LIN {X 0,Y 720.16,Z 195.522,A -85,B 0,C 180,E1 33617.616,E2 33617.616} C_VEL
LIN {X 0,Y 720.211,Z 195.516,A -85,B 0,C 180,E1 33614.811,E2 33614.811} C_VEL
LIN {X 0,Y 720.216,Z 195.521,A -85,B 0,C 180,E1 33611.789,E2 33611.789} C_VEL
LIN {X 0,Y 720.148,Z 195.522,A -85,B 0,C 180,E1 33609.077,E2 33609.077} C_VEL
LIN {X 0,Y 720.178,Z 195.522,A -85,B 0,C 180,E1 33605.959,E2 33605.959} C_VEL
LIN {X 0,Y 720.238,Z 195.651,A -85,B 0,C 180,E1 33604.404,E2 33604.404} C_VEL
LIN {X 0,Y 723.958,Z 206.616,A -85,B 0,C 180,E1 33603.441,E2 33603.441} C_VEL
LIN {X 0,Y 723.246,Z 247.825,A -85,B 0,C 180,E1 33600.537,E2 33600.537} C_VEL
LIN {X 0,Y 722.668,Z 288.727,A -85,B 0,C 180,E1 33597.748,E2 33597.748} C_VEL
LIN {X 0,Y 722.544,Z 304.623,A -85,B 0,C 180,E1 33596.701,E2 33596.701} C_VEL
LIN {X 0,Y 723.876,Z 312.314,A -85,B 0,C 180,E1 33596.564,E2 33596.564} C_VEL
LIN {X 0,Y 722.993,Z 604.896,A -85,B 0,C 180,E1 33593.438,E2 33593.438} C_VEL
LIN {X 0,Y 722.818,Z 626.619,A -85,B 0,C 180,E1 33593.09,E2 33593.09} C_VEL
LIN {X 0,Y 722.561,Z 650.13,A -85,B 0,C 180,E1 33592.539,E2 33592.539} C_VEL
LIN {X 0,Y 722.316,Z 669.51,A -85,B 0,C 180,E1 33591.948,E2 33591.948} C_VEL
LIN {X 0,Y 722.014,Z 689.697,A -85,B 0,C 180,E1 33591.189,E2 33591.189} C_VEL
LIN {X 0,Y 721.715,Z 710.059,A -85,B 0,C 180,E1 33590.265,E2 33590.265} C_VEL
LIN {X 0,Y 721.363,Z 729.936,A -85,B 0,C 180,E1 33589.178,E2 33589.178} C_VEL
LIN {X 0,Y 721.062,Z 746.81,A -85,B 0,C 180,E1 33588.097,E2 33588.097} C_VEL
LIN {X 0,Y 720.802,Z 763.918,A -85,B 0,C 180,E1 33586.83,E2 33586.83} C_VEL
LIN {X 0,Y 720.546,Z 779.819,A -85,B 0,C 180,E1 33585.452,E2 33585.452} C_VEL
LIN {X 0,Y 720.356,Z 792.902,A -85,B 0,C 180,E1 33584.14,E2 33584.14} C_VEL
LIN {X 0,Y 720.195,Z 806.207,A -85,B 0,C 180,E1 33582.59,E2 33582.59} C_VEL
LIN {X 0,Y 720.072,Z 817.974,A -85,B 0,C 180,E1 33580.965,E2 33580.965} C_VEL
LIN {X 0,Y 719.998,Z 827.271,A -85,B 0,C 180,E1 33579.432,E2 33579.432} C_VEL
LIN {X 0,Y 719.944,Z 835.631,A -85,B 0,C 180,E1 33577.742,E2 33577.742} C_VEL
LIN {X 0,Y 719.927,Z 842.505,A -85,B 0,C 180,E1 33575.979,E2 33575.979} C_VEL
LIN {X 0,Y 719.92,Z 847.512,A -85,B 0,C 180,E1 33574.221,E2 33574.221} C_VEL
LIN {X 0,Y 719.914,Z 850.607,A -85,B 0,C 180,E1 33572.547,E2 33572.547} C_VEL
LIN {X 0,Y 719.914,Z 852.289,A -85,B 0,C 180,E1 33570.796,E2 33570.796} C_VEL
LIN {X 0,Y 719.909,Z 852.219,A -85,B 0,C 180,E1 33568.965,E2 33568.965} C_VEL
LIN {X 0,Y 719.913,Z 850.51,A -85,B 0,C 180,E1 33567.293,E2 33567.293} C_VEL
LIN {X 0,Y 719.919,Z 847.147,A -85,B 0,C 180,E1 33565.539,E2 33565.539} C_VEL
LIN {X 0,Y 719.936,Z 841.735,A -85,B 0,C 180,E1 33563.701,E2 33563.701} C_VEL
LIN {X 0,Y 719.958,Z 834.828,A -85,B 0,C 180,E1 33561.985,E2 33561.985} C_VEL
LIN {X 0,Y 720.007,Z 826.408,A -85,B 0,C 180,E1 33560.326,E2 33560.326} C_VEL
LIN {X 0,Y 720.103,Z 815.862,A -85,B 0,C 180,E1 33558.628,E2 33558.628} C_VEL
LIN {X 0,Y 720.228,Z 804.11,A -85,B 0,C 180,E1 33557.056,E2 33557.056} C_VEL
LIN {X 0,Y 720.377,Z 791.433,A -85,B 0,C 180,E1 33555.614,E2 33555.614} C_VEL
LIN {X 0,Y 720.595,Z 776.326,A -85,B 0,C 180,E1 33554.136,E2 33554.136} C_VEL
LIN {X 0,Y 720.851,Z 759.998,A -85,B 0,C 180,E1 33552.774,E2 33552.774} C_VEL
LIN {X 0,Y 721.109,Z 744.471,A -85,B 0,C 180,E1 33551.654,E2 33551.654} C_VEL
LIN {X 0,Y 721.411,Z 726.463,A -85,B 0,C 180,E1 33550.529,E2 33550.529} C_VEL
LIN {X 0,Y 721.75,Z 706.47,A -85,B 0,C 180,E1 33549.474,E2 33549.474} C_VEL
LIN {X 0,Y 722.033,Z 688.563,A -85,B 0,C 180,E1 33548.675,E2 33548.675} C_VEL
LIN {X 0,Y 722.331,Z 668.395,A -85,B 0,C 180,E1 33547.925,E2 33547.925} C_VEL
LIN {X 0,Y 722.629,Z 645.716,A -85,B 0,C 180,E1 33547.254,E2 33547.254} C_VEL
LIN {X 0,Y 722.835,Z 624.224,A -85,B 0,C 180,E1 33546.776,E2 33546.776} C_VEL
LIN {X 0,Y 723.001,Z 603.601,A -85,B 0,C 180,E1 33546.455,E2 33546.455} C_VEL
LIN {X 0,Y 723.876,Z 312.433,A -85,B 0,C 180,E1 33543.347,E2 33543.347} C_VEL
LIN {X 0,Y 722.906,Z 306.324,A -85,B 0,C 180,E1 33543.242,E2 33543.242} C_VEL
LIN {X 0,Y 722.485,Z 303.913,A -85,B 0,C 180,E1 33543.181,E2 33543.181} C_VEL
LIN {X 0,Y 723.04,Z 261.674,A -85,B 0,C 180,E1 33540.325,E2 33540.325} C_VEL
LIN {X 0,Y 723.666,Z 220.838,A -85,B 0,C 180,E1 33537.488,E2 33537.488} C_VEL
LIN {X 0,Y 723.746,Z 206.018,A -85,B 0,C 180,E1 33536.416,E2 33536.416} C_VEL
LIN {X 0,Y 720.207,Z 195.519,A -85,B 0,C 180,E1 33535.473,E2 33535.473} C_VEL
LIN {X 0,Y 720.201,Z 195.524,A -85,B 0,C 180,E1 33532.548,E2 33532.548} C_VEL
LIN {X 0,Y 720.212,Z 195.511,A -85,B 0,C 180,E1 33529.478,E2 33529.478} C_VEL
LIN {X 0,Y 720.206,Z 195.521,A -85,B 0,C 180,E1 33526.479,E2 33526.479} C_VEL
LIN {X 0,Y 720.215,Z 195.509,A -85,B 0,C 180,E1 33523.411,E2 33523.411} C_VEL
LIN {X 0,Y 720.219,Z 195.519,A -85,B 0,C 180,E1 33520.343,E2 33520.343} C_VEL
LIN {X 0,Y 720.208,Z 195.509,A -85,B 0,C 180,E1 33517.252,E2 33517.252} C_VEL
LIN {X 0,Y 720.216,Z 195.521,A -85,B 0,C 180,E1 33514.305,E2 33514.305} C_VEL
LIN {X 0,Y 720.211,Z 195.51,A -85,B 0,C 180,E1 33511.217,E2 33511.217} C_VEL
LIN {X 0,Y 720.217,Z 195.517,A -85,B 0,C 180,E1 33508.166,E2 33508.166} C_VEL
LIN {X 0,Y 720.211,Z 195.51,A -85,B 0,C 180,E1 33505.14,E2 33505.14} C_VEL
LIN {X 0,Y 720.212,Z 195.52,A -85,B 0,C 180,E1 33502.101,E2 33502.101} C_VEL
LIN {X 0,Y 720.215,Z 195.507,A -85,B 0,C 180,E1 33499.126,E2 33499.126} C_VEL
LIN {X 0,Y 720.214,Z 195.52,A -85,B 0,C 180,E1 33496.112,E2 33496.112} C_VEL
LIN {X 0,Y 720.219,Z 195.506,A -85,B 0,C 180,E1 33493.079,E2 33493.079} C_VEL
LIN {X 0,Y 720.212,Z 195.52,A -85,B 0,C 180,E1 33490.075,E2 33490.075} C_VEL
LIN {X 0,Y 720.222,Z 195.506,A -85,B 0,C 180,E1 33487.098,E2 33487.098} C_VEL
LIN {X 0,Y 720.211,Z 195.521,A -85,B 0,C 180,E1 33484.06,E2 33484.06} C_VEL
LIN {X 0,Y 720.219,Z 195.508,A -85,B 0,C 180,E1 33481.034,E2 33481.034} C_VEL
LIN {X 0,Y 720.207,Z 195.52,A -85,B 0,C 180,E1 33478.011,E2 33478.011} C_VEL
LIN {X 0,Y 720.21,Z 195.51,A -85,B 0,C 180,E1 33475.062,E2 33475.062} C_VEL
LIN {X 0,Y 720.201,Z 195.518,A -85,B 0,C 180,E1 33471.939,E2 33471.939} C_VEL
LIN {X 0,Y 720.214,Z 195.51,A -85,B 0,C 180,E1 33468.954,E2 33468.954} C_VEL
LIN {X 0,Y 720.202,Z 195.52,A -85,B 0,C 180,E1 33465.939,E2 33465.939} C_VEL
LIN {X 0,Y 720.196,Z 195.512,A -85,B 0,C 180,E1 33463.049,E2 33463.049} C_VEL
LIN {X 0,Y 720.203,Z 195.521,A -85,B 0,C 180,E1 33459.945,E2 33459.945} C_VEL
LIN {X 0,Y 720.184,Z 195.514,A -85,B 0,C 180,E1 33457.123,E2 33457.123} C_VEL
LIN {X 0,Y 720.218,Z 195.522,A -85,B 0,C 180,E1 33454.109,E2 33454.109} C_VEL
LIN {X 0,Y 720.171,Z 195.516,A -85,B 0,C 180,E1 33451.289,E2 33451.289} C_VEL
LIN {X 0,Y 720.219,Z 195.515,A -85,B 0,C 180,E1 33448.44,E2 33448.44} C_VEL
LIN {X 0,Y 720.171,Z 195.519,A -85,B 0,C 180,E1 33445.559,E2 33445.559} C_VEL
LIN {X 0,Y 720.191,Z 195.514,A -85,B 0,C 180,E1 33442.837,E2 33442.837} C_VEL
LIN {X 0,Y 720.188,Z 195.522,A -85,B 0,C 180,E1 33439.783,E2 33439.783} C_VEL
LIN {X 0,Y 720.163,Z 195.518,A -85,B 0,C 180,E1 33437.131,E2 33437.131} C_VEL
LIN {X 0,Y 720.222,Z 195.518,A -85,B 0,C 180,E1 33434.244,E2 33434.244} C_VEL
LIN {X 0,Y 720.158,Z 195.522,A -85,B 0,C 180,E1 33431.368,E2 33431.368} C_VEL
LIN {X 0,Y 720.209,Z 195.663,A -85,B 0,C 180,E1 33429.793,E2 33429.793} C_VEL
LIN {X 0,Y 721.281,Z 198.701,A -85,B 0,C 180,E1 33429.577,E2 33429.577} C_VEL
LIN {X 0,Y 726.57,Z 209.646,A -85,B 0,C 180,E1 33428.712,E2 33428.712} C_VEL
LIN {X 0,Y 725.859,Z 260.94,A -85,B 0,C 180,E1 33426.323,E2 33426.323} C_VEL
LIN {X 0,Y 725.458,Z 299.229,A -85,B 0,C 180,E1 33424.598,E2 33424.598} C_VEL
LIN {X 0,Y 726.47,Z 307.17,A -85,B 0,C 180,E1 33424.45,E2 33424.45} C_VEL
LIN {X 0,Y 725.424,Z 570.263,A -85,B 0,C 180,E1 33421.465,E2 33421.465} C_VEL
LIN {X 0,Y 724.936,Z 690.96,A -85,B 0,C 180,E1 33420.101,E2 33420.101} C_VEL
LIN {X 0,Y 724.634,Z 716.508,A -85,B 0,C 180,E1 33419.668,E2 33419.668} C_VEL
LIN {X 0,Y 724.35,Z 738.123,A -85,B 0,C 180,E1 33419.168,E2 33419.168} C_VEL
LIN {X 0,Y 724.01,Z 761.286,A -85,B 0,C 180,E1 33418.499,E2 33418.499} C_VEL
LIN {X 0,Y 723.566,Z 783.363,A -85,B 0,C 180,E1 33417.711,E2 33417.711} C_VEL
LIN {X 0,Y 723.176,Z 805.236,A -85,B 0,C 180,E1 33416.791,E2 33416.791} C_VEL
LIN {X 0,Y 722.679,Z 827.148,A -85,B 0,C 180,E1 33415.706,E2 33415.706} C_VEL
LIN {X 0,Y 722.248,Z 847.62,A -85,B 0,C 180,E1 33414.54,E2 33414.54} C_VEL
LIN {X 0,Y 721.793,Z 867.842,A -85,B 0,C 180,E1 33413.211,E2 33413.211} C_VEL
LIN {X 0,Y 721.414,Z 886.71,A -85,B 0,C 180,E1 33411.805,E2 33411.805} C_VEL
LIN {X 0,Y 721.029,Z 904.462,A -85,B 0,C 180,E1 33410.285,E2 33410.285} C_VEL
LIN {X 0,Y 720.755,Z 920.964,A -85,B 0,C 180,E1 33408.691,E2 33408.691} C_VEL
LIN {X 0,Y 720.478,Z 935.22,A -85,B 0,C 180,E1 33407.111,E2 33407.111} C_VEL
LIN {X 0,Y 720.304,Z 948.442,A -85,B 0,C 180,E1 33405.458,E2 33405.458} C_VEL
LIN {X 0,Y 720.157,Z 960.276,A -85,B 0,C 180,E1 33403.734,E2 33403.734} C_VEL
LIN {X 0,Y 720.066,Z 970.03,A -85,B 0,C 180,E1 33402.104,E2 33402.104} C_VEL
LIN {X 0,Y 719.982,Z 980.182,A -85,B 0,C 180,E1 33400.078,E2 33400.078} C_VEL
LIN {X 0,Y 719.928,Z 986.815,A -85,B 0,C 180,E1 33398.466,E2 33398.466} C_VEL
LIN {X 0,Y 719.913,Z 993.245,A -85,B 0,C 180,E1 33396.54,E2 33396.54} C_VEL
LIN {X 0,Y 719.916,Z 997.813,A -85,B 0,C 180,E1 33394.62,E2 33394.62} C_VEL
LIN {X 0,Y 719.882,Z 1000.685,A -85,B 0,C 180,E1 33392.866,E2 33392.866} C_VEL
LIN {X 0,Y 719.891,Z 1002.262,A -85,B 0,C 180,E1 33390.875,E2 33390.875} C_VEL
LIN {X 0,Y 719.883,Z 1002.306,A -85,B 0,C 180,E1 33389.284,E2 33389.284} C_VEL
LIN {X 0,Y 719.888,Z 1001.017,A -85,B 0,C 180,E1 33387.373,E2 33387.373} C_VEL
LIN {X 0,Y 719.917,Z 997.971,A -85,B 0,C 180,E1 33385.459,E2 33385.459} C_VEL
LIN {X 0,Y 719.915,Z 993.864,A -85,B 0,C 180,E1 33383.701,E2 33383.701} C_VEL
LIN {X 0,Y 719.936,Z 987.422,A -85,B 0,C 180,E1 33381.695,E2 33381.695} C_VEL
LIN {X 0,Y 719.968,Z 980.892,A -85,B 0,C 180,E1 33380.084,E2 33380.084} C_VEL
LIN {X 0,Y 720.053,Z 971.867,A -85,B 0,C 180,E1 33378.221,E2 33378.221} C_VEL
LIN {X 0,Y 720.143,Z 961.081,A -85,B 0,C 180,E1 33376.392,E2 33376.392} C_VEL
LIN {X 0,Y 720.295,Z 949.06,A -85,B 0,C 180,E1 33374.625,E2 33374.625} C_VEL
LIN {X 0,Y 720.472,Z 935.927,A -85,B 0,C 180,E1 33372.972,E2 33372.972} C_VEL
LIN {X 0,Y 720.739,Z 921.74,A -85,B 0,C 180,E1 33371.393,E2 33371.393} C_VEL
LIN {X 0,Y 721.008,Z 905.39,A -85,B 0,C 180,E1 33369.799,E2 33369.799} C_VEL
LIN {X 0,Y 721.376,Z 888.27,A -85,B 0,C 180,E1 33368.322,E2 33368.322} C_VEL
LIN {X 0,Y 721.76,Z 869.107,A -85,B 0,C 180,E1 33366.879,E2 33366.879} C_VEL
LIN {X 0,Y 722.231,Z 849.066,A -85,B 0,C 180,E1 33365.547,E2 33365.547} C_VEL
LIN {X 0,Y 722.653,Z 827.944,A -85,B 0,C 180,E1 33364.337,E2 33364.337} C_VEL
LIN {X 0,Y 723.165,Z 806.229,A -85,B 0,C 180,E1 33363.253,E2 33363.253} C_VEL
LIN {X 0,Y 723.547,Z 784.481,A -85,B 0,C 180,E1 33362.333,E2 33362.333} C_VEL
LIN {X 0,Y 723.972,Z 762.568,A -85,B 0,C 180,E1 33361.544,E2 33361.544} C_VEL
LIN {X 0,Y 724.349,Z 738.334,A -85,B 0,C 180,E1 33360.838,E2 33360.838} C_VEL
LIN {X 0,Y 724.63,Z 716.764,A -85,B 0,C 180,E1 33360.337,E2 33360.337} C_VEL
LIN {X 0,Y 724.936,Z 691.166,A -85,B 0,C 180,E1 33359.902,E2 33359.902} C_VEL
LIN {X 0,Y 725.376,Z 582.637,A -85,B 0,C 180,E1 33358.674,E2 33358.674} C_VEL
LIN {X 0,Y 726.451,Z 311.994,A -85,B 0,C 180,E1 33355.606,E2 33355.606} C_VEL
LIN {X 0,Y 726.227,Z 304.001,A -85,B 0,C 180,E1 33355.5,E2 33355.5} C_VEL
LIN {X 0,Y 725.36,Z 298.429,A -85,B 0,C 180,E1 33355.382,E2 33355.382} C_VEL
LIN {X 0,Y 726.223,Z 237.623,A -85,B 0,C 180,E1 33352.602,E2 33352.602} C_VEL
LIN {X 0,Y 726.566,Z 209.659,A -85,B 0,C 180,E1 33351.288,E2 33351.288} C_VEL
LIN {X 0,Y 721.385,Z 198.876,A -85,B 0,C 180,E1 33350.413,E2 33350.413} C_VEL
LIN {X 0,Y 720.172,Z 195.526,A -85,B 0,C 180,E1 33350.156,E2 33350.156} C_VEL
LIN {X 0,Y 720.211,Z 195.521,A -85,B 0,C 180,E1 33347.142,E2 33347.142} C_VEL
LIN {X 0,Y 720.177,Z 195.524,A -85,B 0,C 180,E1 33344.296,E2 33344.296} C_VEL
LIN {X 0,Y 720.221,Z 195.519,A -85,B 0,C 180,E1 33341.316,E2 33341.316} C_VEL
LIN {X 0,Y 720.195,Z 195.524,A -85,B 0,C 180,E1 33338.332,E2 33338.332} C_VEL
LIN {X 0,Y 720.223,Z 195.521,A -85,B 0,C 180,E1 33335.375,E2 33335.375} C_VEL
LIN {X 0,Y 720.201,Z 195.528,A -85,B 0,C 180,E1 33333.906,E2 33333.906} C_VEL
LIN {X 0,Y 724.343,Z 207.121,A -85,B 0,C 180,E1 33332.948,E2 33332.948} C_VEL
LIN {X 0,Y 723.304,Z 257.17,A -85,B 0,C 180,E1 33330.074,E2 33330.074} C_VEL
LIN {X 0,Y 722.6,Z 315.269,A -85,B 0,C 180,E1 33326.859,E2 33326.859} C_VEL
LIN {X 0,Y 722.176,Z 369.58,A -85,B 0,C 180,E1 33323.933,E2 33323.933} C_VEL
LIN {X 0,Y 721.73,Z 424.416,A -85,B 0,C 180,E1 33321.028,E2 33321.028} C_VEL
LIN {X 0,Y 721.364,Z 470.562,A -85,B 0,C 180,E1 33318.625,E2 33318.625} C_VEL
LIN {X 0,Y 721.822,Z 478.064,A -85,B 0,C 180,E1 33318.535,E2 33318.535} C_VEL
LIN {X 0,Y 721.438,Z 679.938,A -85,B 0,C 180,E1 33316.459,E2 33316.459} C_VEL
LIN {X 0,Y 721.316,Z 699.052,A -85,B 0,C 180,E1 33316.11,E2 33316.11} C_VEL
LIN {X 0,Y 721.167,Z 717.241,A -85,B 0,C 180,E1 33315.629,E2 33315.629} C_VEL
LIN {X 0,Y 720.969,Z 734.998,A -85,B 0,C 180,E1 33315.008,E2 33315.008} C_VEL
LIN {X 0,Y 720.803,Z 751.994,A -85,B 0,C 180,E1 33314.254,E2 33314.254} C_VEL
LIN {X 0,Y 720.617,Z 767.716,A -85,B 0,C 180,E1 33313.398,E2 33313.398} C_VEL
LIN {X 0,Y 720.432,Z 783.102,A -85,B 0,C 180,E1 33312.382,E2 33312.382} C_VEL
LIN {X 0,Y 720.274,Z 796.852,A -85,B 0,C 180,E1 33311.288,E2 33311.288} C_VEL
LIN {X 0,Y 720.145,Z 809.523,A -85,B 0,C 180,E1 33310.076,E2 33310.076} C_VEL
LIN {X 0,Y 720.05,Z 820.643,A -85,B 0,C 180,E1 33308.786,E2 33308.786} C_VEL
LIN {X 0,Y 719.983,Z 830.232,A -85,B 0,C 180,E1 33307.421,E2 33307.421} C_VEL
LIN {X 0,Y 719.946,Z 837.854,A -85,B 0,C 180,E1 33306.059,E2 33306.059} C_VEL
LIN {X 0,Y 719.921,Z 844.045,A -85,B 0,C 180,E1 33304.621,E2 33304.621} C_VEL
LIN {X 0,Y 719.914,Z 848.466,A -85,B 0,C 180,E1 33303.185,E2 33303.185} C_VEL
LIN {X 0,Y 719.912,Z 851.34,A -85,B 0,C 180,E1 33301.671,E2 33301.671} C_VEL
LIN {X 0,Y 719.912,Z 852.449,A -85,B 0,C 180,E1 33300.159,E2 33300.159} C_VEL
LIN {X 0,Y 719.913,Z 851.819,A -85,B 0,C 180,E1 33298.647,E2 33298.647} C_VEL
LIN {X 0,Y 719.914,Z 849.435,A -85,B 0,C 180,E1 33297.134,E2 33297.134} C_VEL
LIN {X 0,Y 719.922,Z 845.232,A -85,B 0,C 180,E1 33295.619,E2 33295.619} C_VEL
LIN {X 0,Y 719.936,Z 839.461,A -85,B 0,C 180,E1 33294.181,E2 33294.181} C_VEL
LIN {X 0,Y 719.981,Z 831.802,A -85,B 0,C 180,E1 33292.74,E2 33292.74} C_VEL
LIN {X 0,Y 720.037,Z 822.605,A -85,B 0,C 180,E1 33291.374,E2 33291.374} C_VEL
LIN {X 0,Y 720.131,Z 811.918,A -85,B 0,C 180,E1 33290.086,E2 33290.086} C_VEL
LIN {X 0,Y 720.249,Z 799.731,A -85,B 0,C 180,E1 33288.874,E2 33288.874} C_VEL
LIN {X 0,Y 720.4,Z 785.987,A -85,B 0,C 180,E1 33287.739,E2 33287.739} C_VEL
LIN {X 0,Y 720.572,Z 771.146,A -85,B 0,C 180,E1 33286.721,E2 33286.721} C_VEL
LIN {X 0,Y 720.732,Z 758.498,A -85,B 0,C 180,E1 33285.987,E2 33285.987} C_VEL
LIN {X 0,Y 719.842,Z 752.168,A -85,B 0,C 180,E1 33285.636,E2 33285.636} C_VEL
LIN {X 0,Y 714.42,Z 736.944,A -85,B 0,C 180,E1 33284.836,E2 33284.836} C_VEL
LIN {X 0,Y 713.298,Z 730.158,A -85,B 0,C 180,E1 33284.548,E2 33284.548} C_VEL
LIN {X 0,Y 713.28,Z 729.152,A -85,B 0,C 180,E1 33284.511,E2 33284.511} C_VEL
LIN {X 0,Y 713.505,Z 710.535,A -85,B 0,C 180,E1 33283.911,E2 33283.911} C_VEL
LIN {X 0,Y 713.666,Z 691.674,A -85,B 0,C 180,E1 33283.468,E2 33283.468} C_VEL
LIN {X 0,Y 713.79,Z 672.625,A -85,B 0,C 180,E1 33283.177,E2 33283.177} C_VEL
LIN {X 0,Y 714.094,Z 473.867,A -85,B 0,C 180,E1 33281.121,E2 33281.121} C_VEL
LIN {X 0,Y 713.625,Z 469.588,A -85,B 0,C 180,E1 33281.045,E2 33281.045} C_VEL
LIN {X 0,Y 714.172,Z 418.046,A -85,B 0,C 180,E1 33278.308,E2 33278.308} C_VEL
LIN {X 0,Y 714.783,Z 362.685,A -85,B 0,C 180,E1 33275.319,E2 33275.319} C_VEL
LIN {X 0,Y 715.433,Z 312.1,A -85,B 0,C 180,E1 33272.535,E2 33272.535} C_VEL
LIN {X 0,Y 716.158,Z 259.687,A -85,B 0,C 180,E1 33269.599,E2 33269.599} C_VEL
LIN {X 0,Y 716.883,Z 210.15,A -85,B 0,C 180,E1 33266.76,E2 33266.76} C_VEL
LIN {X 0,Y 716.315,Z 207.723,A -85,B 0,C 180,E1 33266.589,E2 33266.589} C_VEL
LIN {X 0,Y 712.272,Z 196.512,A -85,B 0,C 180,E1 33265.693,E2 33265.693} C_VEL
LIN {X 0,Y 712.274,Z 196.504,A -85,B 0,C 180,E1 33262.667,E2 33262.667} C_VEL
LIN {X 0,Y 712.208,Z 196.513,A -85,B 0,C 180,E1 33259.773,E2 33259.773} C_VEL
LIN {X 0,Y 712.269,Z 196.511,A -85,B 0,C 180,E1 33257.09,E2 33257.09} C_VEL
LIN {X 0,Y 712.265,Z 196.505,A -85,B 0,C 180,E1 33254.131,E2 33254.131} C_VEL
LIN {X 0,Y 712.235,Z 196.508,A -85,B 0,C 180,E1 33251.286,E2 33251.286} C_VEL
LIN {X 0,Y 712.276,Z 196.512,A -85,B 0,C 180,E1 33248.434,E2 33248.434} C_VEL
LIN {X 0,Y 712.234,Z 196.514,A -85,B 0,C 180,E1 33245.536,E2 33245.536} C_VEL
LIN {X 0,Y 712.28,Z 196.515,A -85,B 0,C 180,E1 33244.793,E2 33244.793} C_VEL
LIN {X 0,Y 716.825,Z 210.095,A -85,B 0,C 180,E1 33243.583,E2 33243.583} C_VEL
LIN {X 0,Y 715.958,Z 248.509,A -85,B 0,C 180,E1 33240.834,E2 33240.834} C_VEL
LIN {X 0,Y 715.265,Z 289.395,A -85,B 0,C 180,E1 33238.015,E2 33238.015} C_VEL
LIN {X 0,Y 715.109,Z 304.617,A -85,B 0,C 180,E1 33237.001,E2 33237.001} C_VEL
LIN {X 0,Y 716.715,Z 313.568,A -85,B 0,C 180,E1 33236.837,E2 33236.837} C_VEL
LIN {X 0,Y 715.65,Z 604.587,A -85,B 0,C 180,E1 33233.698,E2 33233.698} C_VEL
LIN {X 0,Y 715.451,Z 625.147,A -85,B 0,C 180,E1 33233.369,E2 33233.369} C_VEL
LIN {X 0,Y 715.193,Z 647.921,A -85,B 0,C 180,E1 33232.85,E2 33232.85} C_VEL
LIN {X 0,Y 714.824,Z 669.791,A -85,B 0,C 180,E1 33232.18,E2 33232.18} C_VEL
LIN {X 0,Y 714.474,Z 689.691,A -85,B 0,C 180,E1 33231.424,E2 33231.424} C_VEL
LIN {X 0,Y 714.107,Z 710.089,A -85,B 0,C 180,E1 33230.489,E2 33230.489} C_VEL
LIN {X 0,Y 713.674,Z 729.931,A -85,B 0,C 180,E1 33229.393,E2 33229.393} C_VEL
LIN {X 0,Y 713.324,Z 746.817,A -85,B 0,C 180,E1 33228.3,E2 33228.3} C_VEL
LIN {X 0,Y 713.005,Z 763.646,A -85,B 0,C 180,E1 33227.043,E2 33227.043} C_VEL
LIN {X 0,Y 712.691,Z 779.818,A -85,B 0,C 180,E1 33225.627,E2 33225.627} C_VEL
LIN {X 0,Y 712.46,Z 792.9,A -85,B 0,C 180,E1 33224.3,E2 33224.3} C_VEL
LIN {X 0,Y 712.265,Z 806.215,A -85,B 0,C 180,E1 33222.733,E2 33222.733} C_VEL
LIN {X 0,Y 712.105,Z 818.482,A -85,B 0,C 180,E1 33221.009,E2 33221.009} C_VEL
LIN {X 0,Y 712.016,Z 827.705,A -85,B 0,C 180,E1 33219.457,E2 33219.457} C_VEL
LIN {X 0,Y 711.958,Z 835.635,A -85,B 0,C 180,E1 33217.83,E2 33217.83} C_VEL
LIN {X 0,Y 711.934,Z 842.509,A -85,B 0,C 180,E1 33216.047,E2 33216.047} C_VEL
LIN {X 0,Y 711.922,Z 847.507,A -85,B 0,C 180,E1 33214.269,E2 33214.269} C_VEL
LIN {X 0,Y 711.915,Z 850.608,A -85,B 0,C 180,E1 33212.576,E2 33212.576} C_VEL
LIN {X 0,Y 711.914,Z 852.292,A -85,B 0,C 180,E1 33210.805,E2 33210.805} C_VEL
LIN {X 0,Y 711.909,Z 852.214,A -85,B 0,C 180,E1 33208.954,E2 33208.954} C_VEL
LIN {X 0,Y 711.912,Z 850.509,A -85,B 0,C 180,E1 33207.263,E2 33207.263} C_VEL
LIN {X 0,Y 711.919,Z 847.149,A -85,B 0,C 180,E1 33205.489,E2 33205.489} C_VEL
LIN {X 0,Y 711.937,Z 841.731,A -85,B 0,C 180,E1 33203.63,E2 33203.63} C_VEL
LIN {X 0,Y 711.97,Z 834.967,A -85,B 0,C 180,E1 33201.927,E2 33201.927} C_VEL
LIN {X 0,Y 712.034,Z 826.408,A -85,B 0,C 180,E1 33200.217,E2 33200.217} C_VEL
LIN {X 0,Y 712.148,Z 815.858,A -85,B 0,C 180,E1 33198.5,E2 33198.5} C_VEL
LIN {X 0,Y 712.297,Z 804.33,A -85,B 0,C 180,E1 33196.938,E2 33196.938} C_VEL
LIN {X 0,Y 712.49,Z 791.429,A -85,B 0,C 180,E1 33195.451,E2 33195.451} C_VEL
LIN {X 0,Y 712.751,Z 776.122,A -85,B 0,C 180,E1 33193.938,E2 33193.938} C_VEL
LIN {X 0,Y 713.054,Z 760.059,A -85,B 0,C 180,E1 33192.585,E2 33192.585} C_VEL
LIN {X 0,Y 713.377,Z 744.454,A -85,B 0,C 180,E1 33191.448,E2 33191.448} C_VEL
LIN {X 0,Y 713.758,Z 726.057,A -85,B 0,C 180,E1 33190.288,E2 33190.288} C_VEL
LIN {X 0,Y 714.156,Z 705.733,A -85,B 0,C 180,E1 33189.211,E2 33189.211} C_VEL
LIN {X 0,Y 714.511,Z 687.71,A -85,B 0,C 180,E1 33188.405,E2 33188.405} C_VEL
LIN {X 0,Y 714.85,Z 668.384,A -85,B 0,C 180,E1 33187.681,E2 33187.681} C_VEL
LIN {X 0,Y 715.217,Z 645.269,A -85,B 0,C 180,E1 33186.994,E2 33186.994} C_VEL
LIN {X 0,Y 715.465,Z 624.006,A -85,B 0,C 180,E1 33186.52,E2 33186.52} C_VEL
LIN {X 0,Y 715.653,Z 604.059,A -85,B 0,C 180,E1 33186.206,E2 33186.206} C_VEL
LIN {X 0,Y 716.712,Z 314.22,A -85,B 0,C 180,E1 33183.08,E2 33183.08} C_VEL
LIN {X 0,Y 716.168,Z 309.757,A -85,B 0,C 180,E1 33183.008,E2 33183.008} C_VEL
LIN {X 0,Y 715.054,Z 303.905,A -85,B 0,C 180,E1 33182.88,E2 33182.88} C_VEL
LIN {X 0,Y 715.713,Z 262.054,A -85,B 0,C 180,E1 33180.018,E2 33180.018} C_VEL
LIN {X 0,Y 716.51,Z 225.81,A -85,B 0,C 180,E1 33177.446,E2 33177.446} C_VEL
LIN {X 0,Y 716.649,Z 209.27,A -85,B 0,C 180,E1 33176.26,E2 33176.26} C_VEL
LIN {X 0,Y 712.244,Z 196.513,A -85,B 0,C 180,E1 33175.087,E2 33175.087} C_VEL
LIN {X 0,Y 712.279,Z 196.512,A -85,B 0,C 180,E1 33172.217,E2 33172.217} C_VEL
LIN {X 0,Y 712.256,Z 196.503,A -85,B 0,C 180,E1 33169.248,E2 33169.248} C_VEL
LIN {X 0,Y 712.28,Z 196.508,A -85,B 0,C 180,E1 33166.299,E2 33166.299} C_VEL
LIN {X 0,Y 712.26,Z 196.5,A -85,B 0,C 180,E1 33163.232,E2 33163.232} C_VEL
LIN {X 0,Y 712.281,Z 196.507,A -85,B 0,C 180,E1 33160.222,E2 33160.222} C_VEL
LIN {X 0,Y 712.268,Z 196.498,A -85,B 0,C 180,E1 33157.232,E2 33157.232} C_VEL
LIN {X 0,Y 712.277,Z 196.508,A -85,B 0,C 180,E1 33154.225,E2 33154.225} C_VEL
LIN {X 0,Y 712.271,Z 196.5,A -85,B 0,C 180,E1 33151.199,E2 33151.199} C_VEL
LIN {X 0,Y 712.276,Z 196.506,A -85,B 0,C 180,E1 33148.143,E2 33148.143} C_VEL
LIN {X 0,Y 712.269,Z 196.499,A -85,B 0,C 180,E1 33145.084,E2 33145.084} C_VEL
LIN {X 0,Y 712.273,Z 196.509,A -85,B 0,C 180,E1 33142.1,E2 33142.1} C_VEL
LIN {X 0,Y 712.274,Z 196.496,A -85,B 0,C 180,E1 33139.092,E2 33139.092} C_VEL
LIN {X 0,Y 712.27,Z 196.508,A -85,B 0,C 180,E1 33136.055,E2 33136.055} C_VEL
LIN {X 0,Y 712.277,Z 196.495,A -85,B 0,C 180,E1 33133.035,E2 33133.035} C_VEL
LIN {X 0,Y 712.268,Z 196.509,A -85,B 0,C 180,E1 33130.025,E2 33130.025} C_VEL
LIN {X 0,Y 712.279,Z 196.496,A -85,B 0,C 180,E1 33127.015,E2 33127.015} C_VEL
LIN {X 0,Y 712.263,Z 196.508,A -85,B 0,C 180,E1 33123.944,E2 33123.944} C_VEL
LIN {X 0,Y 712.282,Z 196.497,A -85,B 0,C 180,E1 33120.965,E2 33120.965} C_VEL
LIN {X 0,Y 712.26,Z 196.507,A -85,B 0,C 180,E1 33117.908,E2 33117.908} C_VEL
LIN {X 0,Y 712.278,Z 196.499,A -85,B 0,C 180,E1 33114.926,E2 33114.926} C_VEL
LIN {X 0,Y 712.262,Z 196.507,A -85,B 0,C 180,E1 33111.93,E2 33111.93} C_VEL
LIN {X 0,Y 712.271,Z 196.5,A -85,B 0,C 180,E1 33108.994,E2 33108.994} C_VEL
LIN {X 0,Y 712.263,Z 196.509,A -85,B 0,C 180,E1 33105.94,E2 33105.94} C_VEL
LIN {X 0,Y 712.261,Z 196.501,A -85,B 0,C 180,E1 33103.022,E2 33103.022} C_VEL
LIN {X 0,Y 712.258,Z 196.509,A -85,B 0,C 180,E1 33099.883,E2 33099.883} C_VEL
LIN {X 0,Y 712.252,Z 196.503,A -85,B 0,C 180,E1 33097.029,E2 33097.029} C_VEL
LIN {X 0,Y 712.265,Z 196.508,A -85,B 0,C 180,E1 33093.935,E2 33093.935} C_VEL
LIN {X 0,Y 712.238,Z 196.503,A -85,B 0,C 180,E1 33091.123,E2 33091.123} C_VEL
LIN {X 0,Y 712.281,Z 196.508,A -85,B 0,C 180,E1 33088.135,E2 33088.135} C_VEL
LIN {X 0,Y 712.228,Z 196.507,A -85,B 0,C 180,E1 33085.349,E2 33085.349} C_VEL
LIN {X 0,Y 712.281,Z 196.504,A -85,B 0,C 180,E1 33082.48,E2 33082.48} C_VEL
LIN {X 0,Y 712.23,Z 196.51,A -85,B 0,C 180,E1 33079.544,E2 33079.544} C_VEL
LIN {X 0,Y 712.251,Z 196.505,A -85,B 0,C 180,E1 33076.769,E2 33076.769} C_VEL
LIN {X 0,Y 712.24,Z 196.514,A -85,B 0,C 180,E1 33073.686,E2 33073.686} C_VEL
LIN {X 0,Y 712.22,Z 196.51,A -85,B 0,C 180,E1 33071.071,E2 33071.071} C_VEL
LIN {X 0,Y 712.307,Z 196.683,A -85,B 0,C 180,E1 33070.259,E2 33070.259} C_VEL
LIN {X 0,Y 713.368,Z 199.645,A -85,B 0,C 180,E1 33070.043,E2 33070.043} C_VEL
LIN {X 0,Y 719.946,Z 213.509,A -85,B 0,C 180,E1 33068.945,E2 33068.945} C_VEL
LIN {X 0,Y 719.057,Z 267.233,A -85,B 0,C 180,E1 33066.425,E2 33066.425} C_VEL
LIN {X 0,Y 718.641,Z 299.284,A -85,B 0,C 180,E1 33064.973,E2 33064.973} C_VEL
LIN {X 0,Y 719.861,Z 308.443,A -85,B 0,C 180,E1 33064.797,E2 33064.797} C_VEL
LIN {X 0,Y 718.584,Z 572.549,A -85,B 0,C 180,E1 33061.773,E2 33061.773} C_VEL
LIN {X 0,Y 718.004,Z 691.175,A -85,B 0,C 180,E1 33060.419,E2 33060.419} C_VEL
LIN {X 0,Y 717.648,Z 716.767,A -85,B 0,C 180,E1 33059.981,E2 33059.981} C_VEL
LIN {X 0,Y 717.298,Z 738.46,A -85,B 0,C 180,E1 33059.474,E2 33059.474} C_VEL
LIN {X 0,Y 716.853,Z 762.568,A -85,B 0,C 180,E1 33058.765,E2 33058.765} C_VEL
LIN {X 0,Y 716.339,Z 784.486,A -85,B 0,C 180,E1 33057.969,E2 33057.969} C_VEL
LIN {X 0,Y 715.831,Z 807.582,A -85,B 0,C 180,E1 33056.978,E2 33056.978} C_VEL
LIN {X 0,Y 715.246,Z 828.756,A -85,B 0,C 180,E1 33055.904,E2 33055.904} C_VEL
LIN {X 0,Y 714.719,Z 849.755,A -85,B 0,C 180,E1 33054.683,E2 33054.683} C_VEL
LIN {X 0,Y 714.182,Z 869.143,A -85,B 0,C 180,E1 33053.379,E2 33053.379} C_VEL
LIN {X 0,Y 713.72,Z 887.819,A -85,B 0,C 180,E1 33051.961,E2 33051.961} C_VEL
LIN {X 0,Y 713.298,Z 904.462,A -85,B 0,C 180,E1 33050.515,E2 33050.515} C_VEL
LIN {X 0,Y 712.937,Z 920.965,A -85,B 0,C 180,E1 33048.904,E2 33048.904} C_VEL
LIN {X 0,Y 712.616,Z 935.222,A -85,B 0,C 180,E1 33047.305,E2 33047.305} C_VEL
LIN {X 0,Y 712.389,Z 949.06,A -85,B 0,C 180,E1 33045.55,E2 33045.55} C_VEL
LIN {X 0,Y 712.21,Z 960.797,A -85,B 0,C 180,E1 33043.808,E2 33043.808} C_VEL
LIN {X 0,Y 712.093,Z 970.948,A -85,B 0,C 180,E1 33042.077,E2 33042.077} C_VEL
LIN {X 0,Y 711.997,Z 980.538,A -85,B 0,C 180,E1 33040.11,E2 33040.11} C_VEL
LIN {X 0,Y 711.935,Z 987.12,A -85,B 0,C 180,E1 33038.48,E2 33038.48} C_VEL
LIN {X 0,Y 711.916,Z 993.451,A -85,B 0,C 180,E1 33036.532,E2 33036.532} C_VEL
LIN {X 0,Y 711.913,Z 997.814,A -85,B 0,C 180,E1 33034.673,E2 33034.673} C_VEL
LIN {X 0,Y 711.882,Z 1000.685,A -85,B 0,C 180,E1 33032.898,E2 33032.898} C_VEL
LIN {X 0,Y 711.891,Z 1002.262,A -85,B 0,C 180,E1 33030.885,E2 33030.885} C_VEL
LIN {X 0,Y 711.883,Z 1002.306,A -85,B 0,C 180,E1 33029.276,E2 33029.276} C_VEL
LIN {X 0,Y 711.887,Z 1001.017,A -85,B 0,C 180,E1 33027.343,E2 33027.343} C_VEL
LIN {X 0,Y 711.917,Z 997.972,A -85,B 0,C 180,E1 33025.408,E2 33025.408} C_VEL
LIN {X 0,Y 711.915,Z 993.864,A -85,B 0,C 180,E1 33023.63,E2 33023.63} C_VEL
LIN {X 0,Y 711.937,Z 987.423,A -85,B 0,C 180,E1 33021.601,E2 33021.601} C_VEL
LIN {X 0,Y 711.989,Z 980.892,A -85,B 0,C 180,E1 33019.971,E2 33019.971} C_VEL
LIN {X 0,Y 712.085,Z 971.866,A -85,B 0,C 180,E1 33018.088,E2 33018.088} C_VEL
LIN {X 0,Y 712.2,Z 961.318,A -85,B 0,C 180,E1 33016.275,E2 33016.275} C_VEL
LIN {X 0,Y 712.375,Z 949.642,A -85,B 0,C 180,E1 33014.533,E2 33014.533} C_VEL
LIN {X 0,Y 712.602,Z 935.929,A -85,B 0,C 180,E1 33012.778,E2 33012.778} C_VEL
LIN {X 0,Y 712.922,Z 921.741,A -85,B 0,C 180,E1 33011.181,E2 33011.181} C_VEL
LIN {X 0,Y 713.27,Z 905.39,A -85,B 0,C 180,E1 33009.57,E2 33009.57} C_VEL
LIN {X 0,Y 713.688,Z 888.776,A -85,B 0,C 180,E1 33008.119,E2 33008.119} C_VEL
LIN {X 0,Y 714.166,Z 869.652,A -85,B 0,C 180,E1 33006.658,E2 33006.658} C_VEL
LIN {X 0,Y 714.698,Z 850.418,A -85,B 0,C 180,E1 33005.36,E2 33005.36} C_VEL
LIN {X 0,Y 715.218,Z 829.552,A -85,B 0,C 180,E1 33004.139,E2 33004.139} C_VEL
LIN {X 0,Y 715.786,Z 808.975,A -85,B 0,C 180,E1 33003.089,E2 33003.089} C_VEL
LIN {X 0,Y 716.313,Z 785.727,A -85,B 0,C 180,E1 33002.08,E2 33002.08} C_VEL
LIN {X 0,Y 716.771,Z 765.133,A -85,B 0,C 180,E1 33001.322,E2 33001.322} C_VEL
LIN {X 0,Y 717.283,Z 740.116,A -85,B 0,C 180,E1 33000.57,E2 33000.57} C_VEL
LIN {X 0,Y 717.613,Z 718.69,A -85,B 0,C 180,E1 33000.06,E2 33000.06} C_VEL
LIN {X 0,Y 717.992,Z 693.629,A -85,B 0,C 180,E1 32999.614,E2 32999.614} C_VEL
LIN {X 0,Y 718.269,Z 642.02,A -85,B 0,C 180,E1 32999.009,E2 32999.009} C_VEL
LIN {X 0,Y 719.445,Z 392.284,A -85,B 0,C 180,E1 32996.173,E2 32996.173} C_VEL
LIN {X 0,Y 719.68,Z 305.755,A -85,B 0,C 180,E1 32995.161,E2 32995.161} C_VEL
LIN {X 0,Y 718.539,Z 298.171,A -85,B 0,C 180,E1 32994.993,E2 32994.993} C_VEL
LIN {X 0,Y 719.603,Z 236.709,A -85,B 0,C 180,E1 32992.154,E2 32992.154} C_VEL
LIN {X 0,Y 719.965,Z 213.374,A -85,B 0,C 180,E1 32991.054,E2 32991.054} C_VEL
LIN {X 0,Y 713.431,Z 199.808,A -85,B 0,C 180,E1 32989.928,E2 32989.928} C_VEL
LIN {X 0,Y 712.281,Z 196.511,A -85,B 0,C 180,E1 32989.664,E2 32989.664} C_VEL
LIN {X 0,Y 712.279,Z 196.511,A -85,B 0,C 180,E1 32986.76,E2 32986.76} C_VEL
LIN {X 0,Y 712.282,Z 196.51,A -85,B 0,C 180,E1 32983.794,E2 32983.794} C_VEL
LIN {X 0,Y 712.264,Z 196.512,A -85,B 0,C 180,E1 32980.829,E2 32980.829} C_VEL
LIN {X 0,Y 712.28,Z 196.51,A -85,B 0,C 180,E1 32977.914,E2 32977.914} C_VEL
LIN {X 0,Y 712.252,Z 196.514,A -85,B 0,C 180,E1 32974.931,E2 32974.931} C_VEL
LIN {X 0,Y 712.253,Z 196.683,A -85,B 0,C 180,E1 32974.345,E2 32974.345} C_VEL
LIN {X 0,Y 717.389,Z 210.124,A -85,B 0,C 180,E1 32973.166,E2 32973.166} C_VEL
LIN {X 0,Y 716.102,Z 258.891,A -85,B 0,C 180,E1 32970.316,E2 32970.316} C_VEL
LIN {X 0,Y 715.192,Z 315.897,A -85,B 0,C 180,E1 32967.115,E2 32967.115} C_VEL
LIN {X 0,Y 714.624,Z 369.984,A -85,B 0,C 180,E1 32964.163,E2 32964.163} C_VEL
LIN {X 0,Y 714.076,Z 424.961,A -85,B 0,C 180,E1 32961.221,E2 32961.221} C_VEL
LIN {X 0,Y 713.69,Z 470.224,A -85,B 0,C 180,E1 32958.853,E2 32958.853} C_VEL
LIN {X 0,Y 714.267,Z 478.095,A -85,B 0,C 180,E1 32958.747,E2 32958.747} C_VEL
LIN {X 0,Y 713.764,Z 680.017,A -85,B 0,C 180,E1 32956.64,E2 32956.64} C_VEL
LIN {X 0,Y 713.62,Z 699.074,A -85,B 0,C 180,E1 32956.288,E2 32956.288} C_VEL
LIN {X 0,Y 713.437,Z 717.391,A -85,B 0,C 180,E1 32955.799,E2 32955.799} C_VEL
LIN {X 0,Y 713.216,Z 734.446,A -85,B 0,C 180,E1 32955.199,E2 32955.199} C_VEL
LIN {X 0,Y 713.007,Z 751.19,A -85,B 0,C 180,E1 32954.455,E2 32954.455} C_VEL
LIN {X 0,Y 712.784,Z 767.054,A -85,B 0,C 180,E1 32953.59,E2 32953.59} C_VEL
LIN {X 0,Y 712.567,Z 781.997,A -85,B 0,C 180,E1 32952.603,E2 32952.603} C_VEL
LIN {X 0,Y 712.373,Z 795.932,A -85,B 0,C 180,E1 32951.497,E2 32951.497} C_VEL
LIN {X 0,Y 712.209,Z 808.757,A -85,B 0,C 180,E1 32950.271,E2 32950.271} C_VEL
LIN {X 0,Y 712.087,Z 820.011,A -85,B 0,C 180,E1 32948.967,E2 32948.967} C_VEL
LIN {X 0,Y 712.002,Z 829.721,A -85,B 0,C 180,E1 32947.586,E2 32947.586} C_VEL
LIN {X 0,Y 711.952,Z 837.452,A -85,B 0,C 180,E1 32946.208,E2 32946.208} C_VEL
LIN {X 0,Y 711.927,Z 843.746,A -85,B 0,C 180,E1 32944.753,E2 32944.753} C_VEL
LIN {X 0,Y 711.914,Z 848.468,A -85,B 0,C 180,E1 32943.221,E2 32943.221} C_VEL
LIN {X 0,Y 711.913,Z 851.342,A -85,B 0,C 180,E1 32941.69,E2 32941.69} C_VEL
LIN {X 0,Y 711.913,Z 852.449,A -85,B 0,C 180,E1 32940.161,E2 32940.161} C_VEL
LIN {X 0,Y 711.912,Z 851.818,A -85,B 0,C 180,E1 32938.632,E2 32938.632} C_VEL
LIN {X 0,Y 711.915,Z 849.433,A -85,B 0,C 180,E1 32937.102,E2 32937.102} C_VEL
LIN {X 0,Y 711.923,Z 845.485,A -85,B 0,C 180,E1 32935.65,E2 32935.65} C_VEL
LIN {X 0,Y 711.94,Z 839.812,A -85,B 0,C 180,E1 32934.196,E2 32934.196} C_VEL
LIN {X 0,Y 711.987,Z 832.719,A -85,B 0,C 180,E1 32932.82,E2 32932.82} C_VEL
LIN {X 0,Y 712.053,Z 823.755,A -85,B 0,C 180,E1 32931.44,E2 32931.44} C_VEL
LIN {X 0,Y 712.161,Z 813.333,A -85,B 0,C 180,E1 32930.137,E2 32930.137} C_VEL
LIN {X 0,Y 712.307,Z 801.092,A -85,B 0,C 180,E1 32928.876,E2 32928.876} C_VEL
LIN {X 0,Y 712.491,Z 787.609,A -85,B 0,C 180,E1 32927.725,E2 32927.725} C_VEL
LIN {X 0,Y 712.703,Z 772.501,A -85,B 0,C 180,E1 32926.657,E2 32926.657} C_VEL
LIN {X 0,Y 712.932,Z 756.541,A -85,B 0,C 180,E1 32925.727,E2 32925.727} C_VEL
LIN {X 0,Y 713.137,Z 739.631,A -85,B 0,C 180,E1 32924.925,E2 32924.925} C_VEL
LIN {X 0,Y 713.28,Z 729.152,A -85,B 0,C 180,E1 32924.511,E2 32924.511} C_VEL
LIN {X 0,Y 712.665,Z 723.159,A -85,B 0,C 180,E1 32924.281,E2 32924.281} C_VEL
LIN {X 0,Y 707.093,Z 705.636,A -85,B 0,C 180,E1 32923.621,E2 32923.621} C_VEL
LIN {X 0,Y 705.967,Z 698.377,A -85,B 0,C 180,E1 32923.421,E2 32923.421} C_VEL
LIN {X 0,Y 705.952,Z 697.308,A -85,B 0,C 180,E1 32923.397,E2 32923.397} C_VEL
LIN {X 0,Y 706.113,Z 677.939,A -85,B 0,C 180,E1 32923.054,E2 32923.054} C_VEL
LIN {X 0,Y 706.629,Z 474.731,A -85,B 0,C 180,E1 32920.895,E2 32920.895} C_VEL
LIN {X 0,Y 705.964,Z 468.931,A -85,B 0,C 180,E1 32920.795,E2 32920.795} C_VEL
LIN {X 0,Y 706.627,Z 415.892,A -85,B 0,C 180,E1 32917.947,E2 32917.947} C_VEL
LIN {X 0,Y 707.369,Z 358.655,A -85,B 0,C 180,E1 32914.819,E2 32914.819} C_VEL
LIN {X 0,Y 708.094,Z 310.205,A -85,B 0,C 180,E1 32912.125,E2 32912.125} C_VEL
LIN {X 0,Y 708.987,Z 256.994,A -85,B 0,C 180,E1 32909.112,E2 32909.112} C_VEL
LIN {X 0,Y 709.718,Z 212.196,A -85,B 0,C 180,E1 32906.516,E2 32906.516} C_VEL
LIN {X 0,Y 704.332,Z 197.5,A -85,B 0,C 180,E1 32905.35,E2 32905.35} C_VEL
LIN {X 0,Y 704.344,Z 197.496,A -85,B 0,C 180,E1 32902.379,E2 32902.379} C_VEL
LIN {X 0,Y 704.266,Z 197.502,A -85,B 0,C 180,E1 32899.546,E2 32899.546} C_VEL
LIN {X 0,Y 704.345,Z 197.496,A -85,B 0,C 180,E1 32896.711,E2 32896.711} C_VEL
LIN {X 0,Y 704.333,Z 197.499,A -85,B 0,C 180,E1 32893.731,E2 32893.731} C_VEL
LIN {X 0,Y 704.305,Z 197.495,A -85,B 0,C 180,E1 32890.826,E2 32890.826} C_VEL
LIN {X 0,Y 704.268,Z 197.504,A -85,B 0,C 180,E1 32887.728,E2 32887.728} C_VEL
LIN {X 0,Y 704.339,Z 197.652,A -85,B 0,C 180,E1 32885.182,E2 32885.182} C_VEL
LIN {X 0,Y 709.779,Z 213.038,A -85,B 0,C 180,E1 32883.782,E2 32883.782} C_VEL
LIN {X 0,Y 708.933,Z 248.718,A -85,B 0,C 180,E1 32881.22,E2 32881.22} C_VEL
LIN {X 0,Y 708.094,Z 278.852,A -85,B 0,C 180,E1 32879.062,E2 32879.062} C_VEL
LIN {X 0,Y 707.707,Z 304.681,A -85,B 0,C 180,E1 32877.307,E2 32877.307} C_VEL
LIN {X 0,Y 709.572,Z 314.84,A -85,B 0,C 180,E1 32877.116,E2 32877.116} C_VEL
LIN {X 0,Y 708.323,Z 604.176,A -85,B 0,C 180,E1 32873.963,E2 32873.963} C_VEL
LIN {X 0,Y 708.111,Z 623.549,A -85,B 0,C 180,E1 32873.656,E2 32873.656} C_VEL
LIN {X 0,Y 707.825,Z 644.177,A -85,B 0,C 180,E1 32873.198,E2 32873.198} C_VEL
LIN {X 0,Y 707.416,Z 667.036,A -85,B 0,C 180,E1 32872.522,E2 32872.522} C_VEL
LIN {X 0,Y 707.008,Z 686.572,A -85,B 0,C 180,E1 32871.792,E2 32871.792} C_VEL
LIN {X 0,Y 706.609,Z 704.141,A -85,B 0,C 180,E1 32871.008,E2 32871.008} C_VEL
LIN {X 0,Y 706.199,Z 722.741,A -85,B 0,C 180,E1 32870.038,E2 32870.038} C_VEL
LIN {X 0,Y 705.716,Z 742.117,A -85,B 0,C 180,E1 32868.834,E2 32868.834} C_VEL
LIN {X 0,Y 705.32,Z 758.277,A -85,B 0,C 180,E1 32867.661,E2 32867.661} C_VEL
LIN {X 0,Y 704.961,Z 774.409,A -85,B 0,C 180,E1 32866.31,E2 32866.31} C_VEL
LIN {X 0,Y 704.623,Z 790.595,A -85,B 0,C 180,E1 32864.715,E2 32864.715} C_VEL
LIN {X 0,Y 704.384,Z 802.926,A -85,B 0,C 180,E1 32863.295,E2 32863.295} C_VEL
LIN {X 0,Y 704.202,Z 814.074,A -85,B 0,C 180,E1 32861.798,E2 32861.798} C_VEL
LIN {X 0,Y 704.077,Z 824.984,A -85,B 0,C 180,E1 32860.06,E2 32860.06} C_VEL
LIN {X 0,Y 703.991,Z 833.448,A -85,B 0,C 180,E1 32858.412,E2 32858.412} C_VEL
LIN {X 0,Y 703.935,Z 839.935,A -85,B 0,C 180,E1 32856.838,E2 32856.838} C_VEL
LIN {X 0,Y 703.916,Z 845.471,A -85,B 0,C 180,E1 32855.134,E2 32855.134} C_VEL
LIN {X 0,Y 703.903,Z 849.66,A -85,B 0,C 180,E1 32853.257,E2 32853.257} C_VEL
LIN {X 0,Y 703.9,Z 851.844,A -85,B 0,C 180,E1 32851.465,E2 32851.465} C_VEL
LIN {X 0,Y 703.902,Z 852.452,A -85,B 0,C 180,E1 32849.674,E2 32849.674} C_VEL
LIN {X 0,Y 703.911,Z 851.29,A -85,B 0,C 180,E1 32847.802,E2 32847.802} C_VEL
LIN {X 0,Y 703.919,Z 848.414,A -85,B 0,C 180,E1 32846.009,E2 32846.009} C_VEL
LIN {X 0,Y 703.925,Z 843.802,A -85,B 0,C 180,E1 32844.212,E2 32844.212} C_VEL
LIN {X 0,Y 703.954,Z 837.441,A -85,B 0,C 180,E1 32842.409,E2 32842.409} C_VEL
LIN {X 0,Y 704.021,Z 829.494,A -85,B 0,C 180,E1 32840.682,E2 32840.682} C_VEL
LIN {X 0,Y 704.122,Z 820.083,A -85,B 0,C 180,E1 32839.031,E2 32839.031} C_VEL
LIN {X 0,Y 704.287,Z 809.445,A -85,B 0,C 180,E1 32837.454,E2 32837.454} C_VEL
LIN {X 0,Y 704.516,Z 795.925,A -85,B 0,C 180,E1 32835.78,E2 32835.78} C_VEL
LIN {X 0,Y 704.779,Z 782.443,A -85,B 0,C 180,E1 32834.362,E2 32834.362} C_VEL
LIN {X 0,Y 705.124,Z 767.259,A -85,B 0,C 180,E1 32832.973,E2 32832.973} C_VEL
LIN {X 0,Y 705.535,Z 749.3,A -85,B 0,C 180,E1 32831.577,E2 32831.577} C_VEL
LIN {X 0,Y 705.94,Z 732.752,A -85,B 0,C 180,E1 32830.472,E2 32830.472} C_VEL
LIN {X 0,Y 706.371,Z 714.967,A -85,B 0,C 180,E1 32829.448,E2 32829.448} C_VEL
LIN {X 0,Y 706.858,Z 693.799,A -85,B 0,C 180,E1 32828.421,E2 32828.421} C_VEL
LIN {X 0,Y 707.285,Z 673.767,A -85,B 0,C 180,E1 32827.624,E2 32827.624} C_VEL
LIN {X 0,Y 707.599,Z 655.35,A -85,B 0,C 180,E1 32827.023,E2 32827.023} C_VEL
LIN {X 0,Y 707.945,Z 636.235,A -85,B 0,C 180,E1 32826.52,E2 32826.52} C_VEL
LIN {X 0,Y 708.226,Z 614.339,A -85,B 0,C 180,E1 32826.088,E2 32826.088} C_VEL
LIN {X 0,Y 708.439,Z 584.242,A -85,B 0,C 180,E1 32825.717,E2 32825.717} C_VEL
LIN {X 0,Y 709.568,Z 313.73,A -85,B 0,C 180,E1 32822.782,E2 32822.782} C_VEL
LIN {X 0,Y 707.643,Z 303.896,A -85,B 0,C 180,E1 32822.572,E2 32822.572} C_VEL
LIN {X 0,Y 708.447,Z 263.895,A -85,B 0,C 180,E1 32819.791,E2 32819.791} C_VEL
LIN {X 0,Y 709.423,Z 230.579,A -85,B 0,C 180,E1 32817.377,E2 32817.377} C_VEL
LIN {X 0,Y 709.669,Z 212.635,A -85,B 0,C 180,E1 32816.086,E2 32816.086} C_VEL
LIN {X 0,Y 704.312,Z 197.503,A -85,B 0,C 180,E1 32814.704,E2 32814.704} C_VEL
LIN {X 0,Y 704.342,Z 197.493,A -85,B 0,C 180,E1 32811.657,E2 32811.657} C_VEL
LIN {X 0,Y 704.315,Z 197.496,A -85,B 0,C 180,E1 32808.678,E2 32808.678} C_VEL
LIN {X 0,Y 704.337,Z 197.493,A -85,B 0,C 180,E1 32805.684,E2 32805.684} C_VEL
LIN {X 0,Y 704.312,Z 197.494,A -85,B 0,C 180,E1 32802.735,E2 32802.735} C_VEL
LIN {X 0,Y 704.329,Z 197.494,A -85,B 0,C 180,E1 32799.823,E2 32799.823} C_VEL
LIN {X 0,Y 704.314,Z 197.491,A -85,B 0,C 180,E1 32796.907,E2 32796.907} C_VEL
LIN {X 0,Y 704.33,Z 197.492,A -85,B 0,C 180,E1 32793.997,E2 32793.997} C_VEL
LIN {X 0,Y 704.321,Z 197.491,A -85,B 0,C 180,E1 32791.02,E2 32791.02} C_VEL
LIN {X 0,Y 704.336,Z 197.494,A -85,B 0,C 180,E1 32788.12,E2 32788.12} C_VEL
LIN {X 0,Y 704.331,Z 197.488,A -85,B 0,C 180,E1 32785.079,E2 32785.079} C_VEL
LIN {X 0,Y 704.335,Z 197.498,A -85,B 0,C 180,E1 32782.099,E2 32782.099} C_VEL
LIN {X 0,Y 704.334,Z 197.485,A -85,B 0,C 180,E1 32779.057,E2 32779.057} C_VEL
LIN {X 0,Y 704.331,Z 197.497,A -85,B 0,C 180,E1 32776.036,E2 32776.036} C_VEL
LIN {X 0,Y 704.339,Z 197.483,A -85,B 0,C 180,E1 32773.045,E2 32773.045} C_VEL
LIN {X 0,Y 704.326,Z 197.497,A -85,B 0,C 180,E1 32769.974,E2 32769.974} C_VEL
LIN {X 0,Y 704.34,Z 197.484,A -85,B 0,C 180,E1 32767.013,E2 32767.013} C_VEL
LIN {X 0,Y 704.327,Z 197.498,A -85,B 0,C 180,E1 32763.989,E2 32763.989} C_VEL
LIN {X 0,Y 704.342,Z 197.486,A -85,B 0,C 180,E1 32760.976,E2 32760.976} C_VEL
LIN {X 0,Y 704.326,Z 197.497,A -85,B 0,C 180,E1 32757.966,E2 32757.966} C_VEL
LIN {X 0,Y 704.338,Z 197.488,A -85,B 0,C 180,E1 32754.95,E2 32754.95} C_VEL
LIN {X 0,Y 704.322,Z 197.495,A -85,B 0,C 180,E1 32751.921,E2 32751.921} C_VEL
LIN {X 0,Y 704.335,Z 197.489,A -85,B 0,C 180,E1 32748.951,E2 32748.951} C_VEL
LIN {X 0,Y 704.317,Z 197.497,A -85,B 0,C 180,E1 32745.843,E2 32745.843} C_VEL
LIN {X 0,Y 704.333,Z 197.49,A -85,B 0,C 180,E1 32742.911,E2 32742.911} C_VEL
LIN {X 0,Y 704.315,Z 197.497,A -85,B 0,C 180,E1 32739.819,E2 32739.819} C_VEL
LIN {X 0,Y 704.324,Z 197.491,A -85,B 0,C 180,E1 32736.916,E2 32736.916} C_VEL
LIN {X 0,Y 704.313,Z 197.496,A -85,B 0,C 180,E1 32733.796,E2 32733.796} C_VEL
LIN {X 0,Y 704.314,Z 197.491,A -85,B 0,C 180,E1 32730.953,E2 32730.953} C_VEL
LIN {X 0,Y 704.311,Z 197.499,A -85,B 0,C 180,E1 32727.793,E2 32727.793} C_VEL
LIN {X 0,Y 704.301,Z 197.494,A -85,B 0,C 180,E1 32725.001,E2 32725.001} C_VEL
LIN {X 0,Y 704.332,Z 197.497,A -85,B 0,C 180,E1 32721.966,E2 32721.966} C_VEL
LIN {X 0,Y 704.286,Z 197.496,A -85,B 0,C 180,E1 32719.175,E2 32719.175} C_VEL
LIN {X 0,Y 704.345,Z 197.495,A -85,B 0,C 180,E1 32716.263,E2 32716.263} C_VEL
LIN {X 0,Y 704.283,Z 197.501,A -85,B 0,C 180,E1 32713.372,E2 32713.372} C_VEL
LIN {X 0,Y 704.318,Z 197.608,A -85,B 0,C 180,E1 32710.764,E2 32710.764} C_VEL
LIN {X 0,Y 705.292,Z 200.424,A -85,B 0,C 180,E1 32710.546,E2 32710.546} C_VEL
LIN {X 0,Y 706.704,Z 203.245,A -85,B 0,C 180,E1 32710.305,E2 32710.305} C_VEL
LIN {X 0,Y 713.285,Z 217.385,A -85,B 0,C 180,E1 32709.176,E2 32709.176} C_VEL
LIN {X 0,Y 712.298,Z 270.275,A -85,B 0,C 180,E1 32706.682,E2 32706.682} C_VEL
LIN {X 0,Y 711.848,Z 299.334,A -85,B 0,C 180,E1 32705.356,E2 32705.356} C_VEL
LIN {X 0,Y 713.279,Z 309.701,A -85,B 0,C 180,E1 32705.15,E2 32705.15} C_VEL
LIN {X 0,Y 711.77,Z 574.266,A -85,B 0,C 180,E1 32702.093,E2 32702.093} C_VEL
LIN {X 0,Y 711.095,Z 691.218,A -85,B 0,C 180,E1 32700.746,E2 32700.746} C_VEL
LIN {X 0,Y 710.694,Z 716.763,A -85,B 0,C 180,E1 32700.305,E2 32700.305} C_VEL
LIN {X 0,Y 710.27,Z 738.453,A -85,B 0,C 180,E1 32699.795,E2 32699.795} C_VEL
LIN {X 0,Y 709.758,Z 762.564,A -85,B 0,C 180,E1 32699.08,E2 32699.08} C_VEL
LIN {X 0,Y 709.159,Z 784.49,A -85,B 0,C 180,E1 32698.278,E2 32698.278} C_VEL
LIN {X 0,Y 708.561,Z 807.17,A -85,B 0,C 180,E1 32697.298,E2 32697.298} C_VEL
LIN {X 0,Y 707.877,Z 828.76,A -85,B 0,C 180,E1 32696.194,E2 32696.194} C_VEL
LIN {X 0,Y 707.237,Z 849.752,A -85,B 0,C 180,E1 32694.962,E2 32694.962} C_VEL
LIN {X 0,Y 706.624,Z 869.053,A -85,B 0,C 180,E1 32693.651,E2 32693.651} C_VEL
LIN {X 0,Y 706.064,Z 887.763,A -85,B 0,C 180,E1 32692.217,E2 32692.217} C_VEL
LIN {X 0,Y 705.564,Z 904.786,A -85,B 0,C 180,E1 32690.719,E2 32690.719} C_VEL
LIN {X 0,Y 705.127,Z 920.967,A -85,B 0,C 180,E1 32689.121,E2 32689.121} C_VEL
LIN {X 0,Y 704.764,Z 935.224,A -85,B 0,C 180,E1 32687.504,E2 32687.504} C_VEL
LIN {X 0,Y 704.49,Z 949.061,A -85,B 0,C 180,E1 32685.729,E2 32685.729} C_VEL
LIN {X 0,Y 704.274,Z 960.798,A -85,B 0,C 180,E1 32683.967,E2 32683.967} C_VEL
LIN {X 0,Y 704.126,Z 971.406,A -85,B 0,C 180,E1 32682.132,E2 32682.132} C_VEL
LIN {X 0,Y 704.018,Z 980.722,A -85,B 0,C 180,E1 32680.183,E2 32680.183} C_VEL
LIN {X 0,Y 703.942,Z 987.424,A -85,B 0,C 180,E1 32678.495,E2 32678.495} C_VEL
LIN {X 0,Y 703.916,Z 993.864,A -85,B 0,C 180,E1 32676.443,E2 32676.443} C_VEL
LIN {X 0,Y 703.915,Z 997.973,A -85,B 0,C 180,E1 32674.644,E2 32674.644} C_VEL
LIN {X 0,Y 703.884,Z 1000.91,A -85,B 0,C 180,E1 32672.768,E2 32672.768} C_VEL
LIN {X 0,Y 703.888,Z 1002.284,A -85,B 0,C 180,E1 32670.814,E2 32670.814} C_VEL
LIN {X 0,Y 703.888,Z 1002.284,A -85,B 0,C 180,E1 32669.186,E2 32669.186} C_VEL
LIN {X 0,Y 703.884,Z 1000.909,A -85,B 0,C 180,E1 32667.232,E2 32667.232} C_VEL
LIN {X 0,Y 703.916,Z 997.972,A -85,B 0,C 180,E1 32665.356,E2 32665.356} C_VEL
LIN {X 0,Y 703.917,Z 993.864,A -85,B 0,C 180,E1 32663.557,E2 32663.557} C_VEL
LIN {X 0,Y 703.94,Z 987.423,A -85,B 0,C 180,E1 32661.505,E2 32661.505} C_VEL
LIN {X 0,Y 704.019,Z 980.721,A -85,B 0,C 180,E1 32659.816,E2 32659.816} C_VEL
LIN {X 0,Y 704.126,Z 971.406,A -85,B 0,C 180,E1 32657.868,E2 32657.868} C_VEL
LIN {X 0,Y 704.275,Z 960.8,A -85,B 0,C 180,E1 32656.033,E2 32656.033} C_VEL
LIN {X 0,Y 704.504,Z 948.438,A -85,B 0,C 180,E1 32654.187,E2 32654.187} C_VEL
LIN {X 0,Y 704.764,Z 935.223,A -85,B 0,C 180,E1 32652.496,E2 32652.496} C_VEL
LIN {X 0,Y 705.146,Z 920.174,A -85,B 0,C 180,E1 32650.793,E2 32650.793} C_VEL
LIN {X 0,Y 705.602,Z 903.533,A -85,B 0,C 180,E1 32649.164,E2 32649.164} C_VEL
LIN {X 0,Y 706.116,Z 885.605,A -85,B 0,C 180,E1 32647.61,E2 32647.61} C_VEL
LIN {X 0,Y 706.66,Z 868.004,A -85,B 0,C 180,E1 32646.274,E2 32646.274} C_VEL
LIN {X 0,Y 707.288,Z 847.62,A -85,B 0,C 180,E1 32644.906,E2 32644.906} C_VEL
LIN {X 0,Y 707.909,Z 827.83,A -85,B 0,C 180,E1 32643.755,E2 32643.755} C_VEL
LIN {X 0,Y 708.585,Z 806.236,A -85,B 0,C 180,E1 32642.657,E2 32642.657} C_VEL
LIN {X 0,Y 709.159,Z 784.489,A -85,B 0,C 180,E1 32641.722,E2 32641.722} C_VEL
LIN {X 0,Y 709.757,Z 762.561,A -85,B 0,C 180,E1 32640.92,E2 32640.92} C_VEL
LIN {X 0,Y 710.273,Z 738.223,A -85,B 0,C 180,E1 32640.199,E2 32640.199} C_VEL
LIN {X 0,Y 710.707,Z 716.369,A -85,B 0,C 180,E1 32639.687,E2 32639.687} C_VEL
LIN {X 0,Y 711.096,Z 691.06,A -85,B 0,C 180,E1 32639.252,E2 32639.252} C_VEL
LIN {X 0,Y 711.957,Z 541.029,A -85,B 0,C 180,E1 32637.528,E2 32637.528} C_VEL
LIN {X 0,Y 713.246,Z 308.067,A -85,B 0,C 180,E1 32634.829,E2 32634.829} C_VEL
LIN {X 0,Y 711.737,Z 298.171,A -85,B 0,C 180,E1 32634.609,E2 32634.609} C_VEL
LIN {X 0,Y 712.953,Z 237.759,A -85,B 0,C 180,E1 32631.794,E2 32631.794} C_VEL
LIN {X 0,Y 713.036,Z 216.483,A -85,B 0,C 180,E1 32630.785,E2 32630.785} C_VEL
LIN {X 0,Y 705.587,Z 200.909,A -85,B 0,C 180,E1 32629.424,E2 32629.424} C_VEL
LIN {X 0,Y 704.305,Z 197.503,A -85,B 0,C 180,E1 32629.12,E2 32629.12} C_VEL
LIN {X 0,Y 704.31,Z 197.502,A -85,B 0,C 180,E1 32626.373,E2 32626.373} C_VEL
LIN {X 0,Y 704.336,Z 197.497,A -85,B 0,C 180,E1 32623.377,E2 32623.377} C_VEL
LIN {X 0,Y 704.295,Z 197.503,A -85,B 0,C 180,E1 32620.451,E2 32620.451} C_VEL
LIN {X 0,Y 704.343,Z 197.497,A -85,B 0,C 180,E1 32617.48,E2 32617.48} C_VEL
LIN {X 0,Y 704.326,Z 197.661,A -85,B 0,C 180,E1 32614.841,E2 32614.841} C_VEL
LIN {X 0,Y 705.506,Z 200.851,A -85,B 0,C 180,E1 32614.535,E2 32614.535} C_VEL
LIN {X 0,Y 710.491,Z 213.304,A -85,B 0,C 180,E1 32613.385,E2 32613.385} C_VEL
LIN {X 0,Y 708.907,Z 262.138,A -85,B 0,C 180,E1 32610.481,E2 32610.481} C_VEL
LIN {X 0,Y 707.787,Z 319.047,A -85,B 0,C 180,E1 32607.24,E2 32607.24} C_VEL
LIN {X 0,Y 707.075,Z 372.246,A -85,B 0,C 180,E1 32604.3,E2 32604.3} C_VEL
LIN {X 0,Y 706.42,Z 427.117,A -85,B 0,C 180,E1 32601.332,E2 32601.332} C_VEL
LIN {X 0,Y 706.013,Z 467.654,A -85,B 0,C 180,E1 32599.193,E2 32599.193} C_VEL
LIN {X 0,Y 707.031,Z 478.159,A -85,B 0,C 180,E1 32599.023,E2 32599.023} C_VEL
LIN {X 0,Y 706.228,Z 638.86,A -85,B 0,C 180,E1 32597.284,E2 32597.284} C_VEL
LIN {X 0,Y 706.078,Z 681.387,A -85,B 0,C 180,E1 32596.805,E2 32596.805} C_VEL
LIN {X 0,Y 705.91,Z 700.233,A -85,B 0,C 180,E1 32596.444,E2 32596.444} C_VEL
LIN {X 0,Y 705.703,Z 718.075,A -85,B 0,C 180,E1 32595.955,E2 32595.955} C_VEL
LIN {X 0,Y 705.433,Z 735.675,A -85,B 0,C 180,E1 32595.319,E2 32595.319} C_VEL
LIN {X 0,Y 705.18,Z 752.818,A -85,B 0,C 180,E1 32594.535,E2 32594.535} C_VEL
LIN {X 0,Y 704.907,Z 769.061,A -85,B 0,C 180,E1 32593.619,E2 32593.619} C_VEL
LIN {X 0,Y 704.65,Z 784.222,A -85,B 0,C 180,E1 32592.581,E2 32592.581} C_VEL
LIN {X 0,Y 704.43,Z 797.789,A -85,B 0,C 180,E1 32591.462,E2 32591.462} C_VEL
LIN {X 0,Y 704.246,Z 810.301,A -85,B 0,C 180,E1 32590.223,E2 32590.223} C_VEL
LIN {X 0,Y 704.107,Z 821.284,A -85,B 0,C 180,E1 32588.905,E2 32588.905} C_VEL
LIN {X 0,Y 704.013,Z 830.753,A -85,B 0,C 180,E1 32587.508,E2 32587.508} C_VEL
LIN {X 0,Y 703.96,Z 838.264,A -85,B 0,C 180,E1 32586.115,E2 32586.115} C_VEL
LIN {X 0,Y 703.926,Z 844.352,A -85,B 0,C 180,E1 32584.644,E2 32584.644} C_VEL
LIN {X 0,Y 703.915,Z 848.674,A -85,B 0,C 180,E1 32583.176,E2 32583.176} C_VEL
LIN {X 0,Y 703.911,Z 851.455,A -85,B 0,C 180,E1 32581.628,E2 32581.628} C_VEL
LIN {X 0,Y 703.916,Z 852.472,A -85,B 0,C 180,E1 32580.081,E2 32580.081} C_VEL
LIN {X 0,Y 703.909,Z 851.748,A -85,B 0,C 180,E1 32578.535,E2 32578.535} C_VEL
LIN {X 0,Y 703.92,Z 849.201,A -85,B 0,C 180,E1 32576.952,E2 32576.952} C_VEL
LIN {X 0,Y 703.924,Z 844.972,A -85,B 0,C 180,E1 32575.438,E2 32575.438} C_VEL
LIN {X 0,Y 703.954,Z 839.101,A -85,B 0,C 180,E1 32573.967,E2 32573.967} C_VEL
LIN {X 0,Y 704.011,Z 831.315,A -85,B 0,C 180,E1 32572.492,E2 32572.492} C_VEL
LIN {X 0,Y 704.104,Z 821.977,A -85,B 0,C 180,E1 32571.095,E2 32571.095} C_VEL
LIN {X 0,Y 704.234,Z 811.14,A -85,B 0,C 180,E1 32569.777,E2 32569.777} C_VEL
LIN {X 0,Y 704.415,Z 798.793,A -85,B 0,C 180,E1 32568.538,E2 32568.538} C_VEL
LIN {X 0,Y 704.628,Z 785.421,A -85,B 0,C 180,E1 32567.419,E2 32567.419} C_VEL
LIN {X 0,Y 704.88,Z 770.501,A -85,B 0,C 180,E1 32566.38,E2 32566.38} C_VEL
LIN {X 0,Y 705.151,Z 754.561,A -85,B 0,C 180,E1 32565.464,E2 32565.464} C_VEL
LIN {X 0,Y 705.4,Z 737.341,A -85,B 0,C 180,E1 32564.66,E2 32564.66} C_VEL
LIN {X 0,Y 705.688,Z 719.079,A -85,B 0,C 180,E1 32563.988,E2 32563.988} C_VEL
LIN {X 0,Y 705.901,Z 700.559,A -85,B 0,C 180,E1 32563.474,E2 32563.474} C_VEL
LIN {X 0,Y 705.952,Z 697.308,A -85,B 0,C 180,E1 32563.397,E2 32563.397} C_VEL
LIN {X 0,Y 705.12,Z 689.881,A -85,B 0,C 180,E1 32563.224,E2 32563.224} C_VEL
LIN {X 0,Y 699.513,Z 671.284,A -85,B 0,C 180,E1 32562.799,E2 32562.799} C_VEL
LIN {X 0,Y 698.559,Z 663.716,A -85,B 0,C 180,E1 32562.688,E2 32562.688} C_VEL
LIN {X 0,Y 699.205,Z 475.631,A -85,B 0,C 180,E1 32560.661,E2 32560.661} C_VEL
LIN {X 0,Y 698.318,Z 468.147,A -85,B 0,C 180,E1 32560.533,E2 32560.533} C_VEL
LIN {X 0,Y 699.133,Z 412.338,A -85,B 0,C 180,E1 32557.503,E2 32557.503} C_VEL
LIN {X 0,Y 699.946,Z 357.952,A -85,B 0,C 180,E1 32554.495,E2 32554.495} C_VEL
LIN {X 0,Y 700.769,Z 309.425,A -85,B 0,C 180,E1 32551.771,E2 32551.771} C_VEL
LIN {X 0,Y 701.828,Z 255.192,A -85,B 0,C 180,E1 32548.667,E2 32548.667} C_VEL
LIN {X 0,Y 702.54,Z 215.212,A -85,B 0,C 180,E1 32546.327,E2 32546.327} C_VEL
LIN {X 0,Y 696.388,Z 198.488,A -85,B 0,C 180,E1 32544.975,E2 32544.975} C_VEL
LIN {X 0,Y 696.382,Z 198.488,A -85,B 0,C 180,E1 32541.977,E2 32541.977} C_VEL
LIN {X 0,Y 696.341,Z 198.491,A -85,B 0,C 180,E1 32539.206,E2 32539.206} C_VEL
LIN {X 0,Y 696.374,Z 198.485,A -85,B 0,C 180,E1 32536.121,E2 32536.121} C_VEL
LIN {X 0,Y 696.382,Z 198.485,A -85,B 0,C 180,E1 32533.227,E2 32533.227} C_VEL
LIN {X 0,Y 696.407,Z 198.487,A -85,B 0,C 180,E1 32530.196,E2 32530.196} C_VEL
LIN {X 0,Y 696.335,Z 198.493,A -85,B 0,C 180,E1 32527.296,E2 32527.296} C_VEL
LIN {X 0,Y 696.386,Z 198.717,A -85,B 0,C 180,E1 32525.603,E2 32525.603} C_VEL
LIN {X 0,Y 702.777,Z 216.31,A -85,B 0,C 180,E1 32523.97,E2 32523.97} C_VEL
LIN {X 0,Y 701.834,Z 254.954,A -85,B 0,C 180,E1 32521.19,E2 32521.19} C_VEL
LIN {X 0,Y 700.991,Z 278.35,A -85,B 0,C 180,E1 32519.479,E2 32519.479} C_VEL
LIN {X 0,Y 700.376,Z 296.666,A -85,B 0,C 180,E1 32518.154,E2 32518.154} C_VEL
LIN {X 0,Y 700.324,Z 304.737,A -85,B 0,C 180,E1 32517.619,E2 32517.619} C_VEL
LIN {X 0,Y 702.442,Z 316.284,A -85,B 0,C 180,E1 32517.398,E2 32517.398} C_VEL
LIN {X 0,Y 701.01,Z 603.766,A -85,B 0,C 180,E1 32514.235,E2 32514.235} C_VEL
LIN {X 0,Y 700.785,Z 622.516,A -85,B 0,C 180,E1 32513.938,E2 32513.938} C_VEL
LIN {X 0,Y 700.461,Z 642.006,A -85,B 0,C 180,E1 32513.512,E2 32513.512} C_VEL
LIN {X 0,Y 700.045,Z 664.513,A -85,B 0,C 180,E1 32512.862,E2 32512.862} C_VEL
LIN {X 0,Y 699.549,Z 684.387,A -85,B 0,C 180,E1 32512.13,E2 32512.13} C_VEL
LIN {X 0,Y 699.109,Z 702.07,A -85,B 0,C 180,E1 32511.346,E2 32511.346} C_VEL
LIN {X 0,Y 698.667,Z 718.036,A -85,B 0,C 180,E1 32510.526,E2 32510.526} C_VEL
LIN {X 0,Y 698.192,Z 736.124,A -85,B 0,C 180,E1 32509.449,E2 32509.449} C_VEL
LIN {X 0,Y 697.638,Z 755.555,A -85,B 0,C 180,E1 32508.077,E2 32508.077} C_VEL
LIN {X 0,Y 697.214,Z 771.068,A -85,B 0,C 180,E1 32506.797,E2 32506.797} C_VEL
LIN {X 0,Y 696.867,Z 784.942,A -85,B 0,C 180,E1 32505.479,E2 32505.479} C_VEL
LIN {X 0,Y 696.552,Z 799.52,A -85,B 0,C 180,E1 32503.87,E2 32503.87} C_VEL
LIN {X 0,Y 696.312,Z 811.743,A -85,B 0,C 180,E1 32502.27,E2 32502.27} C_VEL
LIN {X 0,Y 696.144,Z 821.645,A -85,B 0,C 180,E1 32500.749,E2 32500.749} C_VEL
LIN {X 0,Y 696.03,Z 831.1,A -85,B 0,C 180,E1 32499.009,E2 32499.009} C_VEL
LIN {X 0,Y 695.962,Z 838.667,A -85,B 0,C 180,E1 32497.263,E2 32497.263} C_VEL
LIN {X 0,Y 695.924,Z 844.024,A -85,B 0,C 180,E1 32495.69,E2 32495.69} C_VEL
LIN {X 0,Y 695.918,Z 848.562,A -85,B 0,C 180,E1 32493.872,E2 32493.872} C_VEL
LIN {X 0,Y 695.917,Z 851.512,A -85,B 0,C 180,E1 32491.894,E2 32491.894} C_VEL
LIN {X 0,Y 695.913,Z 852.449,A -85,B 0,C 180,E1 32490.082,E2 32490.082} C_VEL
LIN {X 0,Y 695.906,Z 851.784,A -85,B 0,C 180,E1 32488.353,E2 32488.353} C_VEL
LIN {X 0,Y 695.907,Z 849.522,A -85,B 0,C 180,E1 32486.54,E2 32486.54} C_VEL
LIN {X 0,Y 695.924,Z 845.248,A -85,B 0,C 180,E1 32484.641,E2 32484.641} C_VEL
LIN {X 0,Y 695.943,Z 839.908,A -85,B 0,C 180,E1 32482.985,E2 32482.985} C_VEL
LIN {X 0,Y 696.003,Z 833.105,A -85,B 0,C 180,E1 32481.324,E2 32481.324} C_VEL
LIN {X 0,Y 696.131,Z 823.641,A -85,B 0,C 180,E1 32479.489,E2 32479.489} C_VEL
LIN {X 0,Y 696.282,Z 812.959,A -85,B 0,C 180,E1 32477.813,E2 32477.813} C_VEL
LIN {X 0,Y 696.493,Z 801.626,A -85,B 0,C 180,E1 32476.298,E2 32476.298} C_VEL
LIN {X 0,Y 696.818,Z 787.532,A -85,B 0,C 180,E1 32474.691,E2 32474.691} C_VEL
LIN {X 0,Y 697.194,Z 772.08,A -85,B 0,C 180,E1 32473.203,E2 32473.203} C_VEL
LIN {X 0,Y 697.605,Z 756.696,A -85,B 0,C 180,E1 32471.922,E2 32471.922} C_VEL
LIN {X 0,Y 698.113,Z 738.816,A -85,B 0,C 180,E1 32470.636,E2 32470.636} C_VEL
LIN {X 0,Y 698.603,Z 720.712,A -85,B 0,C 180,E1 32469.532,E2 32469.532} C_VEL
LIN {X 0,Y 699.059,Z 703.818,A -85,B 0,C 180,E1 32468.648,E2 32468.648} C_VEL
LIN {X 0,Y 699.505,Z 686.317,A -85,B 0,C 180,E1 32467.861,E2 32467.861} C_VEL
LIN {X 0,Y 699.98,Z 666.792,A -85,B 0,C 180,E1 32467.126,E2 32467.126} C_VEL
LIN {X 0,Y 700.453,Z 642.92,A -85,B 0,C 180,E1 32466.421,E2 32466.421} C_VEL
LIN {X 0,Y 700.777,Z 623.133,A -85,B 0,C 180,E1 32465.983,E2 32465.983} C_VEL
LIN {X 0,Y 701.005,Z 604.319,A -85,B 0,C 180,E1 32465.682,E2 32465.682} C_VEL
LIN {X 0,Y 702.395,Z 324.273,A -85,B 0,C 180,E1 32462.6,E2 32462.6} C_VEL
LIN {X 0,Y 702.223,Z 314.026,A -85,B 0,C 180,E1 32462.477,E2 32462.477} C_VEL
LIN {X 0,Y 700.249,Z 303.888,A -85,B 0,C 180,E1 32462.258,E2 32462.258} C_VEL
LIN {X 0,Y 700.856,Z 281.358,A -85,B 0,C 180,E1 32460.657,E2 32460.657} C_VEL
LIN {X 0,Y 701.642,Z 260.693,A -85,B 0,C 180,E1 32459.134,E2 32459.134} C_VEL
LIN {X 0,Y 702.661,Z 224.057,A -85,B 0,C 180,E1 32456.487,E2 32456.487} C_VEL
LIN {X 0,Y 702.674,Z 215.893,A -85,B 0,C 180,E1 32455.899,E2 32455.899} C_VEL
LIN {X 0,Y 697.029,Z 200.774,A -85,B 0,C 180,E1 32454.481,E2 32454.481} C_VEL
LIN {X 0,Y 696.4,Z 198.489,A -85,B 0,C 180,E1 32454.269,E2 32454.269} C_VEL
LIN {X 0,Y 696.376,Z 198.485,A -85,B 0,C 180,E1 32451.23,E2 32451.23} C_VEL
LIN {X 0,Y 696.405,Z 198.485,A -85,B 0,C 180,E1 32448.298,E2 32448.298} C_VEL
LIN {X 0,Y 696.387,Z 198.482,A -85,B 0,C 180,E1 32445.287,E2 32445.287} C_VEL
LIN {X 0,Y 696.402,Z 198.488,A -85,B 0,C 180,E1 32442.317,E2 32442.317} C_VEL
LIN {X 0,Y 696.393,Z 198.479,A -85,B 0,C 180,E1 32439.286,E2 32439.286} C_VEL
LIN {X 0,Y 696.401,Z 198.484,A -85,B 0,C 180,E1 32436.204,E2 32436.204} C_VEL
LIN {X 0,Y 696.39,Z 198.474,A -85,B 0,C 180,E1 32433.165,E2 32433.165} C_VEL
LIN {X 0,Y 696.402,Z 198.485,A -85,B 0,C 180,E1 32430.168,E2 32430.168} C_VEL
LIN {X 0,Y 696.391,Z 198.476,A -85,B 0,C 180,E1 32427.101,E2 32427.101} C_VEL
LIN {X 0,Y 696.393,Z 198.477,A -85,B 0,C 180,E1 32424.052,E2 32424.052} C_VEL
LIN {X 0,Y 696.394,Z 198.477,A -85,B 0,C 180,E1 32421.036,E2 32421.036} C_VEL
LIN {X 0,Y 696.393,Z 198.478,A -85,B 0,C 180,E1 32418.068,E2 32418.068} C_VEL
LIN {X 0,Y 696.401,Z 198.476,A -85,B 0,C 180,E1 32415.063,E2 32415.063} C_VEL
LIN {X 0,Y 696.389,Z 198.479,A -85,B 0,C 180,E1 32412.017,E2 32412.017} C_VEL
LIN {X 0,Y 696.399,Z 198.477,A -85,B 0,C 180,E1 32409.004,E2 32409.004} C_VEL
LIN {X 0,Y 696.39,Z 198.478,A -85,B 0,C 180,E1 32406.017,E2 32406.017} C_VEL
LIN {X 0,Y 696.4,Z 198.477,A -85,B 0,C 180,E1 32402.963,E2 32402.963} C_VEL
LIN {X 0,Y 696.383,Z 198.475,A -85,B 0,C 180,E1 32399.918,E2 32399.918} C_VEL
LIN {X 0,Y 696.399,Z 198.476,A -85,B 0,C 180,E1 32396.955,E2 32396.955} C_VEL
LIN {X 0,Y 696.381,Z 198.477,A -85,B 0,C 180,E1 32393.901,E2 32393.901} C_VEL
LIN {X 0,Y 696.401,Z 198.475,A -85,B 0,C 180,E1 32390.913,E2 32390.913} C_VEL
LIN {X 0,Y 696.376,Z 198.486,A -85,B 0,C 180,E1 32387.815,E2 32387.815} C_VEL
LIN {X 0,Y 696.402,Z 198.477,A -85,B 0,C 180,E1 32384.852,E2 32384.852} C_VEL
LIN {X 0,Y 696.37,Z 198.485,A -85,B 0,C 180,E1 32381.759,E2 32381.759} C_VEL
LIN {X 0,Y 696.401,Z 198.478,A -85,B 0,C 180,E1 32378.788,E2 32378.788} C_VEL
LIN {X 0,Y 696.37,Z 198.486,A -85,B 0,C 180,E1 32375.751,E2 32375.751} C_VEL
LIN {X 0,Y 696.387,Z 198.477,A -85,B 0,C 180,E1 32372.832,E2 32372.832} C_VEL
LIN {X 0,Y 696.368,Z 198.487,A -85,B 0,C 180,E1 32369.736,E2 32369.736} C_VEL
LIN {X 0,Y 696.37,Z 198.482,A -85,B 0,C 180,E1 32366.932,E2 32366.932} C_VEL
LIN {X 0,Y 696.373,Z 198.489,A -85,B 0,C 180,E1 32363.799,E2 32363.799} C_VEL
LIN {X 0,Y 696.356,Z 198.484,A -85,B 0,C 180,E1 32361.029,E2 32361.029} C_VEL
LIN {X 0,Y 696.395,Z 198.486,A -85,B 0,C 180,E1 32358.003,E2 32358.003} C_VEL
LIN {X 0,Y 696.344,Z 198.486,A -85,B 0,C 180,E1 32355.167,E2 32355.167} C_VEL
LIN {X 0,Y 696.405,Z 198.488,A -85,B 0,C 180,E1 32352.317,E2 32352.317} C_VEL
LIN {X 0,Y 696.35,Z 198.557,A -85,B 0,C 180,E1 32351.283,E2 32351.283} C_VEL
LIN {X 0,Y 697.377,Z 201.538,A -85,B 0,C 180,E1 32351.047,E2 32351.047} C_VEL
LIN {X 0,Y 700.476,Z 207.638,A -85,B 0,C 180,E1 32350.503,E2 32350.503} C_VEL
LIN {X 0,Y 706.642,Z 220.935,A -85,B 0,C 180,E1 32349.428,E2 32349.428} C_VEL
LIN {X 0,Y 705.501,Z 275.624,A -85,B 0,C 180,E1 32346.835,E2 32346.835} C_VEL
LIN {X 0,Y 705.077,Z 299.347,A -85,B 0,C 180,E1 32345.747,E2 32345.747} C_VEL
LIN {X 0,Y 706.724,Z 311.115,A -85,B 0,C 180,E1 32345.507,E2 32345.507} C_VEL
LIN {X 0,Y 704.965,Z 577.94,A -85,B 0,C 180,E1 32342.397,E2 32342.397} C_VEL
LIN {X 0,Y 704.209,Z 691.357,A -85,B 0,C 180,E1 32341.078,E2 32341.078} C_VEL
LIN {X 0,Y 703.76,Z 716.892,A -85,B 0,C 180,E1 32340.632,E2 32340.632} C_VEL
LIN {X 0,Y 703.262,Z 738.672,A -85,B 0,C 180,E1 32340.116,E2 32340.116} C_VEL
LIN {X 0,Y 702.682,Z 762.561,A -85,B 0,C 180,E1 32339.401,E2 32339.401} C_VEL
LIN {X 0,Y 702.004,Z 784.489,A -85,B 0,C 180,E1 32338.593,E2 32338.593} C_VEL
LIN {X 0,Y 701.295,Z 807.166,A -85,B 0,C 180,E1 32337.605,E2 32337.605} C_VEL
LIN {X 0,Y 700.533,Z 828.597,A -85,B 0,C 180,E1 32336.499,E2 32336.499} C_VEL
LIN {X 0,Y 699.773,Z 849.761,A -85,B 0,C 180,E1 32335.246,E2 32335.246} C_VEL
LIN {X 0,Y 699.088,Z 868.771,A -85,B 0,C 180,E1 32333.943,E2 32333.943} C_VEL
LIN {X 0,Y 698.419,Z 887.762,A -85,B 0,C 180,E1 32332.473,E2 32332.473} C_VEL
LIN {X 0,Y 697.857,Z 904.463,A -85,B 0,C 180,E1 32330.99,E2 32330.99} C_VEL
LIN {X 0,Y 697.329,Z 920.969,A -85,B 0,C 180,E1 32329.343,E2 32329.343} C_VEL
LIN {X 0,Y 696.899,Z 935.933,A -85,B 0,C 180,E1 32327.622,E2 32327.622} C_VEL
LIN {X 0,Y 696.577,Z 949.644,A -85,B 0,C 180,E1 32325.827,E2 32325.827} C_VEL
LIN {X 0,Y 696.33,Z 961.319,A -85,B 0,C 180,E1 32324.044,E2 32324.044} C_VEL
LIN {X 0,Y 696.151,Z 972.299,A -85,B 0,C 180,E1 32322.105,E2 32322.105} C_VEL
LIN {X 0,Y 696.03,Z 981.25,A -85,B 0,C 180,E1 32320.177,E2 32320.177} C_VEL
LIN {X 0,Y 695.956,Z 988.333,A -85,B 0,C 180,E1 32318.344,E2 32318.344} C_VEL
LIN {X 0,Y 695.919,Z 994.277,A -85,B 0,C 180,E1 32316.352,E2 32316.352} C_VEL
LIN {X 0,Y 695.917,Z 998.132,A -85,B 0,C 180,E1 32314.615,E2 32314.615} C_VEL
LIN {X 0,Y 695.888,Z 1001.092,A -85,B 0,C 180,E1 32312.635,E2 32312.635} C_VEL
LIN {X 0,Y 695.885,Z 1002.306,A -85,B 0,C 180,E1 32310.741,E2 32310.741} C_VEL
LIN {X 0,Y 695.899,Z 1002.239,A -85,B 0,C 180,E1 32309.012,E2 32309.012} C_VEL
LIN {X 0,Y 695.885,Z 1000.573,A -85,B 0,C 180,E1 32306.952,E2 32306.952} C_VEL
LIN {X 0,Y 695.906,Z 997.814,A -85,B 0,C 180,E1 32305.22,E2 32305.22} C_VEL
LIN {X 0,Y 695.932,Z 993.244,A -85,B 0,C 180,E1 32303.234,E2 32303.234} C_VEL
LIN {X 0,Y 695.946,Z 987.014,A -85,B 0,C 180,E1 32301.294,E2 32301.294} C_VEL
LIN {X 0,Y 696.047,Z 980.184,A -85,B 0,C 180,E1 32299.572,E2 32299.572} C_VEL
LIN {X 0,Y 696.181,Z 970.03,A -85,B 0,C 180,E1 32297.474,E2 32297.474} C_VEL
LIN {X 0,Y 696.357,Z 960.057,A -85,B 0,C 180,E1 32295.75,E2 32295.75} C_VEL
LIN {X 0,Y 696.635,Z 946.833,A -85,B 0,C 180,E1 32293.787,E2 32293.787} C_VEL
LIN {X 0,Y 696.969,Z 933.81,A -85,B 0,C 180,E1 32292.121,E2 32292.121} C_VEL
LIN {X 0,Y 697.43,Z 917.639,A -85,B 0,C 180,E1 32290.311,E2 32290.311} C_VEL
LIN {X 0,Y 697.916,Z 902.605,A -85,B 0,C 180,E1 32288.836,E2 32288.836} C_VEL
LIN {X 0,Y 698.559,Z 883.396,A -85,B 0,C 180,E1 32287.176,E2 32287.176} C_VEL
LIN {X 0,Y 699.193,Z 865.728,A -85,B 0,C 180,E1 32285.837,E2 32285.837} C_VEL
LIN {X 0,Y 699.955,Z 844.715,A -85,B 0,C 180,E1 32284.443,E2 32284.443} C_VEL
LIN {X 0,Y 700.618,Z 826.323,A -85,B 0,C 180,E1 32283.376,E2 32283.376} C_VEL
LIN {X 0,Y 701.397,Z 803.26,A -85,B 0,C 180,E1 32282.215,E2 32282.215} C_VEL
LIN {X 0,Y 702.081,Z 782.227,A -85,B 0,C 180,E1 32281.318,E2 32281.318} C_VEL
LIN {X 0,Y 702.779,Z 759.174,A -85,B 0,C 180,E1 32280.486,E2 32280.486} C_VEL
LIN {X 0,Y 703.313,Z 736.186,A -85,B 0,C 180,E1 32279.819,E2 32279.819} C_VEL
LIN {X 0,Y 703.913,Z 712.037,A -85,B 0,C 180,E1 32279.266,E2 32279.266} C_VEL
LIN {X 0,Y 704.23,Z 688.169,A -85,B 0,C 180,E1 32278.879,E2 32278.879} C_VEL
LIN {X 0,Y 705.761,Z 447.928,A -85,B 0,C 180,E1 32276.096,E2 32276.096} C_VEL
LIN {X 0,Y 706.574,Z 308.693,A -85,B 0,C 180,E1 32274.454,E2 32274.454} C_VEL
LIN {X 0,Y 704.965,Z 298.307,A -85,B 0,C 180,E1 32274.223,E2 32274.223} C_VEL
LIN {X 0,Y 706.162,Z 241.411,A -85,B 0,C 180,E1 32271.567,E2 32271.567} C_VEL
LIN {X 0,Y 706.508,Z 220.477,A -85,B 0,C 180,E1 32270.562,E2 32270.562} C_VEL
LIN {X 0,Y 699.556,Z 205.772,A -85,B 0,C 180,E1 32269.248,E2 32269.248} C_VEL
LIN {X 0,Y 697.91,Z 202.316,A -85,B 0,C 180,E1 32268.903,E2 32268.903} C_VEL
LIN {X 0,Y 696.412,Z 198.761,A -85,B 0,C 180,E1 32268.545,E2 32268.545} C_VEL
LIN {X 0,Y 696.394,Z 198.489,A -85,B 0,C 180,E1 32268.299,E2 32268.299} C_VEL
LIN {X 0,Y 696.4,Z 198.489,A -85,B 0,C 180,E1 32265.288,E2 32265.288} C_VEL
LIN {X 0,Y 696.399,Z 198.488,A -85,B 0,C 180,E1 32262.316,E2 32262.316} C_VEL
LIN {X 0,Y 696.389,Z 198.489,A -85,B 0,C 180,E1 32259.287,E2 32259.287} C_VEL
LIN {X 0,Y 696.38,Z 198.49,A -85,B 0,C 180,E1 32256.341,E2 32256.341} C_VEL
LIN {X 0,Y 696.412,Z 198.548,A -85,B 0,C 180,E1 32255.399,E2 32255.399} C_VEL
LIN {X 0,Y 697.568,Z 201.776,A -85,B 0,C 180,E1 32255.068,E2 32255.068} C_VEL
LIN {X 0,Y 702.995,Z 214.863,A -85,B 0,C 180,E1 32253.769,E2 32253.769} C_VEL
LIN {X 0,Y 703.618,Z 217.425,A -85,B 0,C 180,E1 32253.559,E2 32253.559} C_VEL
LIN {X 0,Y 701.761,Z 265.146,A -85,B 0,C 180,E1 32250.67,E2 32250.67} C_VEL
LIN {X 0,Y 700.403,Z 322.039,A -85,B 0,C 180,E1 32247.381,E2 32247.381} C_VEL
LIN {X 0,Y 699.523,Z 375.312,A -85,B 0,C 180,E1 32244.399,E2 32244.399} C_VEL
LIN {X 0,Y 698.765,Z 430.143,A -85,B 0,C 180,E1 32241.401,E2 32241.401} C_VEL
LIN {X 0,Y 698.363,Z 465.064,A -85,B 0,C 180,E1 32239.54,E2 32239.54} C_VEL
LIN {X 0,Y 699.86,Z 478.846,A -85,B 0,C 180,E1 32239.307,E2 32239.307} C_VEL
LIN {X 0,Y 698.784,Z 614.753,A -85,B 0,C 180,E1 32237.764,E2 32237.764} C_VEL
LIN {X 0,Y 698.463,Z 681.133,A -85,B 0,C 180,E1 32237.011,E2 32237.011} C_VEL
LIN {X 0,Y 698.264,Z 700.156,A -85,B 0,C 180,E1 32236.642,E2 32236.642} C_VEL
LIN {X 0,Y 698.014,Z 718.42,A -85,B 0,C 180,E1 32236.135,E2 32236.135} C_VEL
LIN {X 0,Y 697.708,Z 735.718,A -85,B 0,C 180,E1 32235.502,E2 32235.502} C_VEL
LIN {X 0,Y 697.411,Z 752.149,A -85,B 0,C 180,E1 32234.743,E2 32234.743} C_VEL
LIN {X 0,Y 697.096,Z 767.73,A -85,B 0,C 180,E1 32233.859,E2 32233.859} C_VEL
LIN {X 0,Y 696.804,Z 782.562,A -85,B 0,C 180,E1 32232.851,E2 32232.851} C_VEL
LIN {X 0,Y 696.55,Z 795.949,A -85,B 0,C 180,E1 32231.761,E2 32231.761} C_VEL
LIN {X 0,Y 696.327,Z 808.765,A -85,B 0,C 180,E1 32230.508,E2 32230.508} C_VEL
LIN {X 0,Y 696.159,Z 820.017,A -85,B 0,C 180,E1 32229.174,E2 32229.174} C_VEL
LIN {X 0,Y 696.042,Z 829.727,A -85,B 0,C 180,E1 32227.761,E2 32227.761} C_VEL
LIN {X 0,Y 695.969,Z 837.458,A -85,B 0,C 180,E1 32226.351,E2 32226.351} C_VEL
LIN {X 0,Y 695.935,Z 843.749,A -85,B 0,C 180,E1 32224.863,E2 32224.863} C_VEL
LIN {X 0,Y 695.914,Z 848.47,A -85,B 0,C 180,E1 32223.295,E2 32223.295} C_VEL
LIN {X 0,Y 695.914,Z 851.344,A -85,B 0,C 180,E1 32221.729,E2 32221.729} C_VEL
LIN {X 0,Y 695.915,Z 852.45,A -85,B 0,C 180,E1 32220.165,E2 32220.165} C_VEL
LIN {X 0,Y 695.911,Z 851.815,A -85,B 0,C 180,E1 32218.6,E2 32218.6} C_VEL
LIN {X 0,Y 695.918,Z 849.429,A -85,B 0,C 180,E1 32217.035,E2 32217.035} C_VEL
LIN {X 0,Y 695.927,Z 845.48,A -85,B 0,C 180,E1 32215.55,E2 32215.55} C_VEL
LIN {X 0,Y 695.953,Z 839.807,A -85,B 0,C 180,E1 32214.062,E2 32214.062} C_VEL
LIN {X 0,Y 696.016,Z 832.713,A -85,B 0,C 180,E1 32212.654,E2 32212.654} C_VEL
LIN {X 0,Y 696.111,Z 823.748,A -85,B 0,C 180,E1 32211.242,E2 32211.242} C_VEL
LIN {X 0,Y 696.26,Z 813.325,A -85,B 0,C 180,E1 32209.909,E2 32209.909} C_VEL
LIN {X 0,Y 696.453,Z 801.453,A -85,B 0,C 180,E1 32208.656,E2 32208.656} C_VEL
LIN {X 0,Y 696.7,Z 788.1,A -85,B 0,C 180,E1 32207.484,E2 32207.484} C_VEL
LIN {X 0,Y 696.992,Z 773.136,A -85,B 0,C 180,E1 32206.392,E2 32206.392} C_VEL
LIN {X 0,Y 697.307,Z 757.411,A -85,B 0,C 180,E1 32205.445,E2 32205.445} C_VEL
LIN {X 0,Y 697.602,Z 740.74,A -85,B 0,C 180,E1 32204.623,E2 32204.623} C_VEL
LIN {X 0,Y 697.929,Z 723.561,A -85,B 0,C 180,E1 32203.948,E2 32203.948} C_VEL
LIN {X 0,Y 698.192,Z 705.148,A -85,B 0,C 180,E1 32203.393,E2 32203.393} C_VEL
LIN {X 0,Y 698.405,Z 686.432,A -85,B 0,C 180,E1 32202.99,E2 32202.99} C_VEL
LIN {X 0,Y 698.554,Z 664.873,A -85,B 0,C 180,E1 32202.7,E2 32202.7} C_VEL
LIN {X 0,Y 698.559,Z 663.716,A -85,B 0,C 180,E1 32202.688,E2 32202.688} C_VEL
LIN {X 0,Y 697.628,Z 656.12,A -85,B 0,C 180,E1 32202.578,E2 32202.578} C_VEL
LIN {X 0,Y 691.754,Z 636.216,A -85,B 0,C 180,E1 32202.201,E2 32202.201} C_VEL
LIN {X 0,Y 691.079,Z 629.682,A -85,B 0,C 180,E1 32202.112,E2 32202.112} C_VEL
LIN {X 0,Y 691.757,Z 476.22,A -85,B 0,C 180,E1 32200.415,E2 32200.415} C_VEL
LIN {X 0,Y 690.687,Z 467.362,A -85,B 0,C 180,E1 32200.265,E2 32200.265} C_VEL
LIN {X 0,Y 691.604,Z 411.541,A -85,B 0,C 180,E1 32197.203,E2 32197.203} C_VEL
LIN {X 0,Y 692.526,Z 357.73,A -85,B 0,C 180,E1 32194.194,E2 32194.194} C_VEL
LIN {X 0,Y 693.468,Z 308.718,A -85,B 0,C 180,E1 32191.414,E2 32191.414} C_VEL
LIN {X 0,Y 694.686,Z 254.271,A -85,B 0,C 180,E1 32188.264,E2 32188.264} C_VEL
LIN {X 0,Y 695.434,Z 218.314,A -85,B 0,C 180,E1 32186.14,E2 32186.14} C_VEL
LIN {X 0,Y 688.466,Z 199.475,A -85,B 0,C 180,E1 32184.585,E2 32184.585} C_VEL
LIN {X 0,Y 688.413,Z 199.479,A -85,B 0,C 180,E1 32181.659,E2 32181.659} C_VEL
LIN {X 0,Y 688.459,Z 199.476,A -85,B 0,C 180,E1 32178.748,E2 32178.748} C_VEL
LIN {X 0,Y 688.43,Z 199.476,A -85,B 0,C 180,E1 32175.8,E2 32175.8} C_VEL
LIN {X 0,Y 688.441,Z 199.472,A -85,B 0,C 180,E1 32172.936,E2 32172.936} C_VEL
LIN {X 0,Y 688.433,Z 199.478,A -85,B 0,C 180,E1 32169.926,E2 32169.926} C_VEL
LIN {X 0,Y 688.409,Z 199.483,A -85,B 0,C 180,E1 32167.117,E2 32167.117} C_VEL
LIN {X 0,Y 688.456,Z 199.683,A -85,B 0,C 180,E1 32166.03,E2 32166.03} C_VEL
LIN {X 0,Y 694.615,Z 216.106,A -85,B 0,C 180,E1 32164.501,E2 32164.501} C_VEL
LIN {X 0,Y 695.816,Z 220.075,A -85,B 0,C 180,E1 32164.135,E2 32164.135} C_VEL
LIN {X 0,Y 694.796,Z 259.327,A -85,B 0,C 180,E1 32161.3,E2 32161.3} C_VEL
LIN {X 0,Y 693.822,Z 286.378,A -85,B 0,C 180,E1 32159.321,E2 32159.321} C_VEL
LIN {X 0,Y 693.028,Z 305.154,A -85,B 0,C 180,E1 32157.931,E2 32157.931} C_VEL
LIN {X 0,Y 695.332,Z 317.607,A -85,B 0,C 180,E1 32157.688,E2 32157.688} C_VEL
LIN {X 0,Y 693.715,Z 603.355,A -85,B 0,C 180,E1 32154.512,E2 32154.512} C_VEL
LIN {X 0,Y 693.473,Z 621.628,A -85,B 0,C 180,E1 32154.224,E2 32154.224} C_VEL
LIN {X 0,Y 693.136,Z 640.087,A -85,B 0,C 180,E1 32153.823,E2 32153.823} C_VEL
LIN {X 0,Y 692.732,Z 658.203,A -85,B 0,C 180,E1 32153.319,E2 32153.319} C_VEL
LIN {X 0,Y 692.239,Z 679.129,A -85,B 0,C 180,E1 32152.595,E2 32152.595} C_VEL
LIN {X 0,Y 691.651,Z 699.38,A -85,B 0,C 180,E1 32151.721,E2 32151.721} C_VEL
LIN {X 0,Y 691.114,Z 716.765,A -85,B 0,C 180,E1 32150.832,E2 32150.832} C_VEL
LIN {X 0,Y 690.586,Z 733.368,A -85,B 0,C 180,E1 32149.848,E2 32149.848} C_VEL
LIN {X 0,Y 690.055,Z 750.457,A -85,B 0,C 180,E1 32148.677,E2 32148.677} C_VEL
LIN {X 0,Y 689.512,Z 768.174,A -85,B 0,C 180,E1 32147.251,E2 32147.251} C_VEL
LIN {X 0,Y 689.083,Z 782.384,A -85,B 0,C 180,E1 32145.917,E2 32145.917} C_VEL
LIN {X 0,Y 688.746,Z 795.167,A -85,B 0,C 180,E1 32144.546,E2 32144.546} C_VEL
LIN {X 0,Y 688.435,Z 808.796,A -85,B 0,C 180,E1 32142.839,E2 32142.839} C_VEL
LIN {X 0,Y 688.217,Z 819.525,A -85,B 0,C 180,E1 32141.226,E2 32141.226} C_VEL
LIN {X 0,Y 688.086,Z 828.13,A -85,B 0,C 180,E1 32139.704,E2 32139.704} C_VEL
LIN {X 0,Y 688.002,Z 836.002,A -85,B 0,C 180,E1 32138.02,E2 32138.02} C_VEL
LIN {X 0,Y 687.938,Z 843.277,A -85,B 0,C 180,E1 32136.007,E2 32136.007} C_VEL
LIN {X 0,Y 687.923,Z 847.67,A -85,B 0,C 180,E1 32134.335,E2 32134.335} C_VEL
LIN {X 0,Y 687.912,Z 850.609,A -85,B 0,C 180,E1 32132.666,E2 32132.666} C_VEL
LIN {X 0,Y 687.914,Z 852.301,A -85,B 0,C 180,E1 32130.833,E2 32130.833} C_VEL
LIN {X 0,Y 687.907,Z 852.2,A -85,B 0,C 180,E1 32128.917,E2 32128.917} C_VEL
LIN {X 0,Y 687.909,Z 850.5,A -85,B 0,C 180,E1 32127.167,E2 32127.167} C_VEL
LIN {X 0,Y 687.919,Z 847.327,A -85,B 0,C 180,E1 32125.415,E2 32125.415} C_VEL
LIN {X 0,Y 687.942,Z 842.019,A -85,B 0,C 180,E1 32123.49,E2 32123.49} C_VEL
LIN {X 0,Y 688.006,Z 835.314,A -85,B 0,C 180,E1 32121.728,E2 32121.728} C_VEL
LIN {X 0,Y 688.101,Z 827.283,A -85,B 0,C 180,E1 32120.042,E2 32120.042} C_VEL
LIN {X 0,Y 688.263,Z 817.487,A -85,B 0,C 180,E1 32118.35,E2 32118.35} C_VEL
LIN {X 0,Y 688.502,Z 805.631,A -85,B 0,C 180,E1 32116.649,E2 32116.649} C_VEL
LIN {X 0,Y 688.804,Z 792.928,A -85,B 0,C 180,E1 32115.112,E2 32115.112} C_VEL
LIN {X 0,Y 689.152,Z 779.852,A -85,B 0,C 180,E1 32113.738,E2 32113.738} C_VEL
LIN {X 0,Y 689.655,Z 763.188,A -85,B 0,C 180,E1 32112.23,E2 32112.23} C_VEL
LIN {X 0,Y 690.162,Z 746.849,A -85,B 0,C 180,E1 32110.975,E2 32110.975} C_VEL
LIN {X 0,Y 690.671,Z 730.636,A -85,B 0,C 180,E1 32109.89,E2 32109.89} C_VEL
LIN {X 0,Y 691.266,Z 712.545,A -85,B 0,C 180,E1 32108.845,E2 32108.845} C_VEL
LIN {X 0,Y 691.877,Z 691.767,A -85,B 0,C 180,E1 32107.84,E2 32107.84} C_VEL
LIN {X 0,Y 692.376,Z 673.27,A -85,B 0,C 180,E1 32107.1,E2 32107.1} C_VEL
LIN {X 0,Y 692.771,Z 656.015,A -85,B 0,C 180,E1 32106.525,E2 32106.525} C_VEL
LIN {X 0,Y 693.178,Z 638.161,A -85,B 0,C 180,E1 32106.04,E2 32106.04} C_VEL
LIN {X 0,Y 693.52,Z 618.807,A -85,B 0,C 180,E1 32105.633,E2 32105.633} C_VEL
LIN {X 0,Y 693.807,Z 595.213,A -85,B 0,C 180,E1 32105.294,E2 32105.294} C_VEL
LIN {X 0,Y 695.329,Z 316.439,A -85,B 0,C 180,E1 32102.209,E2 32102.209} C_VEL
LIN {X 0,Y 692.953,Z 304.605,A -85,B 0,C 180,E1 32101.961,E2 32101.961} C_VEL
LIN {X 0,Y 694.338,Z 274.175,A -85,B 0,C 180,E1 32099.686,E2 32099.686} C_VEL
LIN {X 0,Y 695.424,Z 236.86,A -85,B 0,C 180,E1 32096.98,E2 32096.98} C_VEL
LIN {X 0,Y 695.747,Z 219.344,A -85,B 0,C 180,E1 32095.711,E2 32095.711} C_VEL
LIN {X 0,Y 689.56,Z 202.639,A -85,B 0,C 180,E1 32094.139,E2 32094.139} C_VEL
LIN {X 0,Y 688.459,Z 199.475,A -85,B 0,C 180,E1 32093.854,E2 32093.854} C_VEL
LIN {X 0,Y 688.43,Z 199.477,A -85,B 0,C 180,E1 32090.924,E2 32090.924} C_VEL
LIN {X 0,Y 688.456,Z 199.475,A -85,B 0,C 180,E1 32087.968,E2 32087.968} C_VEL
LIN {X 0,Y 688.434,Z 199.474,A -85,B 0,C 180,E1 32084.982,E2 32084.982} C_VEL
LIN {X 0,Y 688.455,Z 199.476,A -85,B 0,C 180,E1 32082.032,E2 32082.032} C_VEL
LIN {X 0,Y 688.44,Z 199.47,A -85,B 0,C 180,E1 32079.076,E2 32079.076} C_VEL
LIN {X 0,Y 688.459,Z 199.474,A -85,B 0,C 180,E1 32076.133,E2 32076.133} C_VEL
LIN {X 0,Y 688.446,Z 199.464,A -85,B 0,C 180,E1 32073.068,E2 32073.068} C_VEL
LIN {X 0,Y 688.455,Z 199.472,A -85,B 0,C 180,E1 32070.071,E2 32070.071} C_VEL
LIN {X 0,Y 688.449,Z 199.466,A -85,B 0,C 180,E1 32067.039,E2 32067.039} C_VEL
LIN {X 0,Y 688.452,Z 199.465,A -85,B 0,C 180,E1 32064,E2 32064} C_VEL
LIN {X 0,Y 688.454,Z 199.467,A -85,B 0,C 180,E1 32061.023,E2 32061.023} C_VEL
LIN {X 0,Y 688.451,Z 199.466,A -85,B 0,C 180,E1 32058.021,E2 32058.021} C_VEL
LIN {X 0,Y 688.456,Z 199.467,A -85,B 0,C 180,E1 32054.982,E2 32054.982} C_VEL
LIN {X 0,Y 688.449,Z 199.467,A -85,B 0,C 180,E1 32051.987,E2 32051.987} C_VEL
LIN {X 0,Y 688.458,Z 199.467,A -85,B 0,C 180,E1 32048.94,E2 32048.94} C_VEL
LIN {X 0,Y 688.444,Z 199.466,A -85,B 0,C 180,E1 32045.919,E2 32045.919} C_VEL
LIN {X 0,Y 688.46,Z 199.467,A -85,B 0,C 180,E1 32042.914,E2 32042.914} C_VEL
LIN {X 0,Y 688.444,Z 199.463,A -85,B 0,C 180,E1 32039.917,E2 32039.917} C_VEL
LIN {X 0,Y 688.461,Z 199.466,A -85,B 0,C 180,E1 32036.92,E2 32036.92} C_VEL
LIN {X 0,Y 688.437,Z 199.464,A -85,B 0,C 180,E1 32033.83,E2 32033.83} C_VEL
LIN {X 0,Y 688.464,Z 199.464,A -85,B 0,C 180,E1 32030.807,E2 32030.807} C_VEL
LIN {X 0,Y 688.433,Z 199.474,A -85,B 0,C 180,E1 32027.757,E2 32027.757} C_VEL
LIN {X 0,Y 688.467,Z 199.466,A -85,B 0,C 180,E1 32024.759,E2 32024.759} C_VEL
LIN {X 0,Y 688.429,Z 199.473,A -85,B 0,C 180,E1 32021.716,E2 32021.716} C_VEL
LIN {X 0,Y 688.461,Z 199.467,A -85,B 0,C 180,E1 32018.799,E2 32018.799} C_VEL
LIN {X 0,Y 688.43,Z 199.475,A -85,B 0,C 180,E1 32015.73,E2 32015.73} C_VEL
LIN {X 0,Y 688.454,Z 199.466,A -85,B 0,C 180,E1 32012.774,E2 32012.774} C_VEL
LIN {X 0,Y 688.429,Z 199.477,A -85,B 0,C 180,E1 32009.735,E2 32009.735} C_VEL
LIN {X 0,Y 688.434,Z 199.471,A -85,B 0,C 180,E1 32006.899,E2 32006.899} C_VEL
LIN {X 0,Y 688.431,Z 199.478,A -85,B 0,C 180,E1 32003.762,E2 32003.762} C_VEL
LIN {X 0,Y 688.425,Z 199.472,A -85,B 0,C 180,E1 32000.923,E2 32000.923} C_VEL
LIN {X 0,Y 688.435,Z 199.479,A -85,B 0,C 180,E1 31997.794,E2 31997.794} C_VEL
LIN {X 0,Y 688.411,Z 199.474,A -85,B 0,C 180,E1 31995.02,E2 31995.02} C_VEL
LIN {X 0,Y 688.462,Z 199.478,A -85,B 0,C 180,E1 31992.031,E2 31992.031} C_VEL
LIN {X 0,Y 688.45,Z 199.58,A -85,B 0,C 180,E1 31991.808,E2 31991.808} C_VEL
LIN {X 0,Y 689.516,Z 202.648,A -85,B 0,C 180,E1 31991.559,E2 31991.559} C_VEL
LIN {X 0,Y 696.062,Z 215.958,A -85,B 0,C 180,E1 31990.38,E2 31990.38} C_VEL
LIN {X 0,Y 700.012,Z 224.6,A -85,B 0,C 180,E1 31989.679,E2 31989.679} C_VEL
LIN {X 0,Y 698.681,Z 280.566,A -85,B 0,C 180,E1 31987.007,E2 31987.007} C_VEL
LIN {X 0,Y 698.335,Z 299.337,A -85,B 0,C 180,E1 31986.147,E2 31986.147} C_VEL
LIN {X 0,Y 700.197,Z 312.41,A -85,B 0,C 180,E1 31985.873,E2 31985.873} C_VEL
LIN {X 0,Y 698.191,Z 580.103,A -85,B 0,C 180,E1 31982.725,E2 31982.725} C_VEL
LIN {X 0,Y 697.348,Z 691.401,A -85,B 0,C 180,E1 31981.417,E2 31981.417} C_VEL
LIN {X 0,Y 696.858,Z 716.759,A -85,B 0,C 180,E1 31980.972,E2 31980.972} C_VEL
LIN {X 0,Y 696.284,Z 738.562,A -85,B 0,C 180,E1 31980.453,E2 31980.453} C_VEL
LIN {X 0,Y 695.63,Z 762.557,A -85,B 0,C 180,E1 31979.729,E2 31979.729} C_VEL
LIN {X 0,Y 694.911,Z 783.354,A -85,B 0,C 180,E1 31978.959,E2 31978.959} C_VEL
LIN {X 0,Y 694.117,Z 805.252,A -85,B 0,C 180,E1 31978.009,E2 31978.009} C_VEL
LIN {X 0,Y 693.259,Z 827.137,A -85,B 0,C 180,E1 31976.882,E2 31976.882} C_VEL
LIN {X 0,Y 692.489,Z 846.179,A -85,B 0,C 180,E1 31975.761,E2 31975.761} C_VEL
LIN {X 0,Y 691.611,Z 867.23,A -85,B 0,C 180,E1 31974.333,E2 31974.333} C_VEL
LIN {X 0,Y 690.896,Z 885.056,A -85,B 0,C 180,E1 31972.956,E2 31972.956} C_VEL
LIN {X 0,Y 690.213,Z 902.605,A -85,B 0,C 180,E1 31971.412,E2 31971.412} C_VEL
LIN {X 0,Y 689.669,Z 917.638,A -85,B 0,C 180,E1 31969.92,E2 31969.92} C_VEL
LIN {X 0,Y 689.134,Z 933.813,A -85,B 0,C 180,E1 31968.089,E2 31968.089} C_VEL
LIN {X 0,Y 688.759,Z 946.529,A -85,B 0,C 180,E1 31966.444,E2 31966.444} C_VEL
LIN {X 0,Y 688.438,Z 959.761,A -85,B 0,C 180,E1 31964.466,E2 31964.466} C_VEL
LIN {X 0,Y 688.231,Z 969.568,A -85,B 0,C 180,E1 31962.758,E2 31962.758} C_VEL
LIN {X 0,Y 688.063,Z 979.475,A -85,B 0,C 180,E1 31960.72,E2 31960.72} C_VEL
LIN {X 0,Y 687.966,Z 986.513,A -85,B 0,C 180,E1 31958.947,E2 31958.947} C_VEL
LIN {X 0,Y 687.931,Z 992.253,A -85,B 0,C 180,E1 31957.181,E2 31957.181} C_VEL
LIN {X 0,Y 687.891,Z 997.338,A -85,B 0,C 180,E1 31955.087,E2 31955.087} C_VEL
LIN {X 0,Y 687.903,Z 1000.236,A -85,B 0,C 180,E1 31953.333,E2 31953.333} C_VEL
LIN {X 0,Y 687.91,Z 1002.171,A -85,B 0,C 180,E1 31951.249,E2 31951.249} C_VEL
LIN {X 0,Y 687.882,Z 1002.351,A -85,B 0,C 180,E1 31949.417,E2 31949.417} C_VEL
LIN {X 0,Y 687.905,Z 1001.296,A -85,B 0,C 180,E1 31947.584,E2 31947.584} C_VEL
LIN {X 0,Y 687.918,Z 998.448,A -85,B 0,C 180,E1 31945.498,E2 31945.498} C_VEL
LIN {X 0,Y 687.924,Z 994.689,A -85,B 0,C 180,E1 31943.742,E2 31943.742} C_VEL
LIN {X 0,Y 687.973,Z 989.148,A -85,B 0,C 180,E1 31941.794,E2 31941.794} C_VEL
LIN {X 0,Y 688.046,Z 981.605,A -85,B 0,C 180,E1 31939.788,E2 31939.788} C_VEL
LIN {X 0,Y 688.162,Z 973.524,A -85,B 0,C 180,E1 31938.008,E2 31938.008} C_VEL
LIN {X 0,Y 688.375,Z 962.356,A -85,B 0,C 180,E1 31935.961,E2 31935.961} C_VEL
LIN {X 0,Y 688.624,Z 951.385,A -85,B 0,C 180,E1 31934.245,E2 31934.245} C_VEL
LIN {X 0,Y 689.012,Z 937.332,A -85,B 0,C 180,E1 31932.344,E2 31932.344} C_VEL
LIN {X 0,Y 689.463,Z 923.3,A -85,B 0,C 180,E1 31930.691,E2 31930.691} C_VEL
LIN {X 0,Y 690.089,Z 906.16,A -85,B 0,C 180,E1 31928.926,E2 31928.926} C_VEL
LIN {X 0,Y 690.7,Z 889.787,A -85,B 0,C 180,E1 31927.441,E2 31927.441} C_VEL
LIN {X 0,Y 691.496,Z 870.26,A -85,B 0,C 180,E1 31925.89,E2 31925.89} C_VEL
LIN {X 0,Y 692.24,Z 851.743,A -85,B 0,C 180,E1 31924.596,E2 31924.596} C_VEL
LIN {X 0,Y 693.127,Z 830.364,A -85,B 0,C 180,E1 31923.297,E2 31923.297} C_VEL
LIN {X 0,Y 693.907,Z 810.763,A -85,B 0,C 180,E1 31922.262,E2 31922.262} C_VEL
LIN {X 0,Y 694.788,Z 786.736,A -85,B 0,C 180,E1 31921.177,E2 31921.177} C_VEL
LIN {X 0,Y 695.479,Z 766.409,A -85,B 0,C 180,E1 31920.406,E2 31920.406} C_VEL
LIN {X 0,Y 696.232,Z 741.99,A -85,B 0,C 180,E1 31919.639,E2 31919.639} C_VEL
LIN {X 0,Y 696.762,Z 719.611,A -85,B 0,C 180,E1 31919.089,E2 31919.089} C_VEL
LIN {X 0,Y 697.321,Z 695.022,A -85,B 0,C 180,E1 31918.632,E2 31918.632} C_VEL
LIN {X 0,Y 697.718,Z 648.066,A -85,B 0,C 180,E1 31918.062,E2 31918.062} C_VEL
LIN {X 0,Y 699.507,Z 400.707,A -85,B 0,C 180,E1 31915.175,E2 31915.175} C_VEL
LIN {X 0,Y 700.021,Z 309.905,A -85,B 0,C 180,E1 31914.085,E2 31914.085} C_VEL
LIN {X 0,Y 698.228,Z 298.171,A -85,B 0,C 180,E1 31913.817,E2 31913.817} C_VEL
LIN {X 0,Y 699.098,Z 250.456,A -85,B 0,C 180,E1 31911.608,E2 31911.608} C_VEL
LIN {X 0,Y 699.861,Z 224.104,A -85,B 0,C 180,E1 31910.31,E2 31910.31} C_VEL
LIN {X 0,Y 693.919,Z 211.305,A -85,B 0,C 180,E1 31909.142,E2 31909.142} C_VEL
LIN {X 0,Y 689.985,Z 203.273,A -85,B 0,C 180,E1 31908.272,E2 31908.272} C_VEL
LIN {X 0,Y 688.566,Z 200.105,A -85,B 0,C 180,E1 31907.906,E2 31907.906} C_VEL
LIN {X 0,Y 688.461,Z 199.476,A -85,B 0,C 180,E1 31907.828,E2 31907.828} C_VEL
LIN {X 0,Y 688.417,Z 199.481,A -85,B 0,C 180,E1 31904.745,E2 31904.745} C_VEL
LIN {X 0,Y 688.446,Z 199.477,A -85,B 0,C 180,E1 31901.921,E2 31901.921} C_VEL
LIN {X 0,Y 688.42,Z 199.481,A -85,B 0,C 180,E1 31898.743,E2 31898.743} C_VEL
LIN {X 0,Y 688.436,Z 199.53,A -85,B 0,C 180,E1 31896.031,E2 31896.031} C_VEL
LIN {X 0,Y 689.691,Z 202.873,A -85,B 0,C 180,E1 31895.648,E2 31895.648} C_VEL
LIN {X 0,Y 693.396,Z 211.165,A -85,B 0,C 180,E1 31894.719,E2 31894.719} C_VEL
LIN {X 0,Y 696.871,Z 220.343,A -85,B 0,C 180,E1 31893.822,E2 31893.822} C_VEL
LIN {X 0,Y 694.716,Z 266.624,A -85,B 0,C 180,E1 31890.962,E2 31890.962} C_VEL
LIN {X 0,Y 693.093,Z 322.938,A -85,B 0,C 180,E1 31887.651,E2 31887.651} C_VEL
LIN {X 0,Y 692.042,Z 375.961,A -85,B 0,C 180,E1 31884.64,E2 31884.64} C_VEL
LIN {X 0,Y 691.144,Z 430.671,A -85,B 0,C 180,E1 31881.61,E2 31881.61} C_VEL
LIN {X 0,Y 690.744,Z 462.706,A -85,B 0,C 180,E1 31879.885,E2 31879.885} C_VEL
LIN {X 0,Y 692.647,Z 479.634,A -85,B 0,C 180,E1 31879.586,E2 31879.586} C_VEL
LIN {X 0,Y 691.201,Z 622.884,A -85,B 0,C 180,E1 31877.896,E2 31877.896} C_VEL
LIN {X 0,Y 690.846,Z 681.611,A -85,B 0,C 180,E1 31877.209,E2 31877.209} C_VEL
LIN {X 0,Y 690.614,Z 700.894,A -85,B 0,C 180,E1 31876.827,E2 31876.827} C_VEL
LIN {X 0,Y 690.343,Z 718.904,A -85,B 0,C 180,E1 31876.319,E2 31876.319} C_VEL
LIN {X 0,Y 690.011,Z 736.238,A -85,B 0,C 180,E1 31875.68,E2 31875.68} C_VEL
LIN {X 0,Y 689.69,Z 752.449,A -85,B 0,C 180,E1 31874.927,E2 31874.927} C_VEL
LIN {X 0,Y 689.339,Z 768.367,A -85,B 0,C 180,E1 31874.019,E2 31874.019} C_VEL
LIN {X 0,Y 688.989,Z 783.057,A -85,B 0,C 180,E1 31873,E2 31873} C_VEL
LIN {X 0,Y 688.669,Z 796.479,A -85,B 0,C 180,E1 31871.876,E2 31871.876} C_VEL
LIN {X 0,Y 688.393,Z 808.805,A -85,B 0,C 180,E1 31870.63,E2 31870.63} C_VEL
LIN {X 0,Y 688.188,Z 820.655,A -85,B 0,C 180,E1 31869.197,E2 31869.197} C_VEL
LIN {X 0,Y 688.057,Z 830.244,A -85,B 0,C 180,E1 31867.767,E2 31867.767} C_VEL
LIN {X 0,Y 687.976,Z 837.865,A -85,B 0,C 180,E1 31866.342,E2 31866.342} C_VEL
LIN {X 0,Y 687.936,Z 844.054,A -85,B 0,C 180,E1 31864.836,E2 31864.836} C_VEL
LIN {X 0,Y 687.915,Z 848.471,A -85,B 0,C 180,E1 31863.333,E2 31863.333} C_VEL
LIN {X 0,Y 687.914,Z 851.344,A -85,B 0,C 180,E1 31861.749,E2 31861.749} C_VEL
LIN {X 0,Y 687.915,Z 852.449,A -85,B 0,C 180,E1 31860.167,E2 31860.167} C_VEL
LIN {X 0,Y 687.911,Z 851.815,A -85,B 0,C 180,E1 31858.584,E2 31858.584} C_VEL
LIN {X 0,Y 687.919,Z 849.427,A -85,B 0,C 180,E1 31857.001,E2 31857.001} C_VEL
LIN {X 0,Y 687.927,Z 845.478,A -85,B 0,C 180,E1 31855.498,E2 31855.498} C_VEL
LIN {X 0,Y 687.961,Z 839.805,A -85,B 0,C 180,E1 31853.993,E2 31853.993} C_VEL
LIN {X 0,Y 688.032,Z 832.71,A -85,B 0,C 180,E1 31852.568,E2 31852.568} C_VEL
LIN {X 0,Y 688.142,Z 823.731,A -85,B 0,C 180,E1 31851.138,E2 31851.138} C_VEL
LIN {X 0,Y 688.311,Z 813.319,A -85,B 0,C 180,E1 31849.792,E2 31849.792} C_VEL
LIN {X 0,Y 688.567,Z 800.725,A -85,B 0,C 180,E1 31848.44,E2 31848.44} C_VEL
LIN {X 0,Y 688.87,Z 787.333,A -85,B 0,C 180,E1 31847.254,E2 31847.254} C_VEL
LIN {X 0,Y 689.204,Z 772.853,A -85,B 0,C 180,E1 31846.193,E2 31846.193} C_VEL
LIN {X 0,Y 689.555,Z 757.405,A -85,B 0,C 180,E1 31845.257,E2 31845.257} C_VEL
LIN {X 0,Y 689.877,Z 741.064,A -85,B 0,C 180,E1 31844.447,E2 31844.447} C_VEL
LIN {X 0,Y 690.236,Z 723.857,A -85,B 0,C 180,E1 31843.765,E2 31843.765} C_VEL
LIN {X 0,Y 690.53,Z 705.346,A -85,B 0,C 180,E1 31843.201,E2 31843.201} C_VEL
LIN {X 0,Y 690.77,Z 686.648,A -85,B 0,C 180,E1 31842.793,E2 31842.793} C_VEL
LIN {X 0,Y 690.94,Z 665.223,A -85,B 0,C 180,E1 31842.5,E2 31842.5} C_VEL
LIN {X 0,Y 691.079,Z 629.682,A -85,B 0,C 180,E1 31842.112,E2 31842.112} C_VEL
LIN {X 0,Y 690.185,Z 622.078,A -85,B 0,C 180,E1 31842.004,E2 31842.004} C_VEL
LIN {X 0,Y 684.349,Z 602.175,A -85,B 0,C 180,E1 31841.618,E2 31841.618} C_VEL
LIN {X 0,Y 683.666,Z 595.646,A -85,B 0,C 180,E1 31841.524,E2 31841.524} C_VEL
LIN {X 0,Y 684.359,Z 477.101,A -85,B 0,C 180,E1 31840.169,E2 31840.169} C_VEL
LIN {X 0,Y 683.081,Z 466.178,A -85,B 0,C 180,E1 31839.969,E2 31839.969} C_VEL
LIN {X 0,Y 684.091,Z 410.724,A -85,B 0,C 180,E1 31836.893,E2 31836.893} C_VEL
LIN {X 0,Y 685.114,Z 357.611,A -85,B 0,C 180,E1 31833.894,E2 31833.894} C_VEL
LIN {X 0,Y 686.192,Z 308.344,A -85,B 0,C 180,E1 31831.067,E2 31831.067} C_VEL
LIN {X 0,Y 687.528,Z 254.78,A -85,B 0,C 180,E1 31827.938,E2 31827.938} C_VEL
LIN {X 0,Y 688.374,Z 221.597,A -85,B 0,C 180,E1 31825.961,E2 31825.961} C_VEL
LIN {X 0,Y 680.517,Z 200.457,A -85,B 0,C 180,E1 31824.2,E2 31824.2} C_VEL
LIN {X 0,Y 680.464,Z 200.468,A -85,B 0,C 180,E1 31821.354,E2 31821.354} C_VEL
LIN {X 0,Y 680.506,Z 200.466,A -85,B 0,C 180,E1 31818.383,E2 31818.383} C_VEL
LIN {X 0,Y 680.516,Z 200.465,A -85,B 0,C 180,E1 31815.385,E2 31815.385} C_VEL
LIN {X 0,Y 680.525,Z 200.46,A -85,B 0,C 180,E1 31812.294,E2 31812.294} C_VEL
LIN {X 0,Y 680.452,Z 200.467,A -85,B 0,C 180,E1 31809.382,E2 31809.382} C_VEL
LIN {X 0,Y 680.535,Z 200.535,A -85,B 0,C 180,E1 31806.464,E2 31806.464} C_VEL
LIN {X 0,Y 686.453,Z 215.886,A -85,B 0,C 180,E1 31805.053,E2 31805.053} C_VEL
LIN {X 0,Y 688.911,Z 223.653,A -85,B 0,C 180,E1 31804.325,E2 31804.325} C_VEL
LIN {X 0,Y 687.771,Z 263.046,A -85,B 0,C 180,E1 31801.461,E2 31801.461} C_VEL
LIN {X 0,Y 686.505,Z 299.257,A -85,B 0,C 180,E1 31798.823,E2 31798.823} C_VEL
LIN {X 0,Y 686.257,Z 307.834,A -85,B 0,C 180,E1 31798.209,E2 31798.209} C_VEL
LIN {X 0,Y 688.261,Z 319.043,A -85,B 0,C 180,E1 31797.986,E2 31797.986} C_VEL
LIN {X 0,Y 686.423,Z 604.169,A -85,B 0,C 180,E1 31794.779,E2 31794.779} C_VEL
LIN {X 0,Y 686.158,Z 621.906,A -85,B 0,C 180,E1 31794.493,E2 31794.493} C_VEL
LIN {X 0,Y 685.806,Z 639.574,A -85,B 0,C 180,E1 31794.107,E2 31794.107} C_VEL
LIN {X 0,Y 685.366,Z 656.998,A -85,B 0,C 180,E1 31793.623,E2 31793.623} C_VEL
LIN {X 0,Y 684.883,Z 675.569,A -85,B 0,C 180,E1 31792.988,E2 31792.988} C_VEL
LIN {X 0,Y 684.193,Z 697.588,A -85,B 0,C 180,E1 31792.06,E2 31792.06} C_VEL
LIN {X 0,Y 683.576,Z 715.679,A -85,B 0,C 180,E1 31791.135,E2 31791.135} C_VEL
LIN {X 0,Y 682.983,Z 731.983,A -85,B 0,C 180,E1 31790.168,E2 31790.168} C_VEL
LIN {X 0,Y 682.442,Z 747.427,A -85,B 0,C 180,E1 31789.115,E2 31789.115} C_VEL
LIN {X 0,Y 681.841,Z 764.705,A -85,B 0,C 180,E1 31787.76,E2 31787.76} C_VEL
LIN {X 0,Y 681.295,Z 780.672,A -85,B 0,C 180,E1 31786.279,E2 31786.279} C_VEL
LIN {X 0,Y 680.919,Z 793.306,A -85,B 0,C 180,E1 31784.93,E2 31784.93} C_VEL
LIN {X 0,Y 680.58,Z 805.591,A -85,B 0,C 180,E1 31783.423,E2 31783.423} C_VEL
LIN {X 0,Y 680.298,Z 817.976,A -85,B 0,C 180,E1 31781.617,E2 31781.617} C_VEL
LIN {X 0,Y 680.127,Z 827.25,A -85,B 0,C 180,E1 31779.99,E2 31779.99} C_VEL
LIN {X 0,Y 680.021,Z 835.299,A -85,B 0,C 180,E1 31778.282,E2 31778.282} C_VEL
LIN {X 0,Y 679.948,Z 842.269,A -85,B 0,C 180,E1 31776.417,E2 31776.417} C_VEL
LIN {X 0,Y 679.918,Z 847.307,A -85,B 0,C 180,E1 31774.555,E2 31774.555} C_VEL
LIN {X 0,Y 679.908,Z 850.487,A -85,B 0,C 180,E1 31772.782,E2 31772.782} C_VEL
LIN {X 0,Y 679.9,Z 852.132,A -85,B 0,C 180,E1 31771.096,E2 31771.096} C_VEL
LIN {X 0,Y 679.91,Z 852.329,A -85,B 0,C 180,E1 31769.157,E2 31769.157} C_VEL
LIN {X 0,Y 679.912,Z 850.73,A -85,B 0,C 180,E1 31767.303,E2 31767.303} C_VEL
LIN {X 0,Y 679.923,Z 847.849,A -85,B 0,C 180,E1 31765.611,E2 31765.611} C_VEL
LIN {X 0,Y 679.948,Z 843.297,A -85,B 0,C 180,E1 31763.838,E2 31763.838} C_VEL
LIN {X 0,Y 680.014,Z 836.027,A -85,B 0,C 180,E1 31761.8,E2 31761.8} C_VEL
LIN {X 0,Y 680.112,Z 828.15,A -85,B 0,C 180,E1 31760.095,E2 31760.095} C_VEL
LIN {X 0,Y 680.263,Z 819.549,A -85,B 0,C 180,E1 31758.555,E2 31758.555} C_VEL
LIN {X 0,Y 680.526,Z 808.194,A -85,B 0,C 180,E1 31756.836,E2 31756.836} C_VEL
LIN {X 0,Y 680.864,Z 795.192,A -85,B 0,C 180,E1 31755.195,E2 31755.195} C_VEL
LIN {X 0,Y 681.219,Z 783.264,A -85,B 0,C 180,E1 31753.894,E2 31753.894} C_VEL
LIN {X 0,Y 681.65,Z 770.12,A -85,B 0,C 180,E1 31752.632,E2 31752.632} C_VEL
LIN {X 0,Y 682.171,Z 755.037,A -85,B 0,C 180,E1 31751.365,E2 31751.365} C_VEL
LIN {X 0,Y 682.874,Z 735.446,A -85,B 0,C 180,E1 31749.963,E2 31749.963} C_VEL
LIN {X 0,Y 683.454,Z 718.898,A -85,B 0,C 180,E1 31748.956,E2 31748.956} C_VEL
LIN {X 0,Y 684.007,Z 702.968,A -85,B 0,C 180,E1 31748.114,E2 31748.114} C_VEL
LIN {X 0,Y 684.517,Z 686.647,A -85,B 0,C 180,E1 31747.367,E2 31747.367} C_VEL
LIN {X 0,Y 685.073,Z 668.594,A -85,B 0,C 180,E1 31746.668,E2 31746.668} C_VEL
LIN {X 0,Y 685.682,Z 646.288,A -85,B 0,C 180,E1 31745.97,E2 31745.97} C_VEL
LIN {X 0,Y 686.107,Z 624.882,A -85,B 0,C 180,E1 31745.474,E2 31745.474} C_VEL
LIN {X 0,Y 686.401,Z 606.327,A -85,B 0,C 180,E1 31745.161,E2 31745.161} C_VEL
LIN {X 0,Y 687.07,Z 504.663,A -85,B 0,C 180,E1 31744.009,E2 31744.009} C_VEL
LIN {X 0,Y 688.092,Z 316.943,A -85,B 0,C 180,E1 31741.892,E2 31741.892} C_VEL
LIN {X 0,Y 686.181,Z 307.3,A -85,B 0,C 180,E1 31741.685,E2 31741.685} C_VEL
LIN {X 0,Y 687.433,Z 274.484,A -85,B 0,C 180,E1 31739.275,E2 31739.275} C_VEL
LIN {X 0,Y 688.659,Z 233.526,A -85,B 0,C 180,E1 31736.301,E2 31736.301} C_VEL
LIN {X 0,Y 688.736,Z 222.447,A -85,B 0,C 180,E1 31735.483,E2 31735.483} C_VEL
LIN {X 0,Y 682.873,Z 206.786,A -85,B 0,C 180,E1 31733.998,E2 31733.998} C_VEL
LIN {X 0,Y 680.513,Z 200.463,A -85,B 0,C 180,E1 31733.435,E2 31733.435} C_VEL
LIN {X 0,Y 680.524,Z 200.466,A -85,B 0,C 180,E1 31730.346,E2 31730.346} C_VEL
LIN {X 0,Y 680.504,Z 200.461,A -85,B 0,C 180,E1 31727.247,E2 31727.247} C_VEL
LIN {X 0,Y 680.522,Z 200.462,A -85,B 0,C 180,E1 31724.26,E2 31724.26} C_VEL
LIN {X 0,Y 680.505,Z 200.46,A -85,B 0,C 180,E1 31721.168,E2 31721.168} C_VEL
LIN {X 0,Y 680.522,Z 200.463,A -85,B 0,C 180,E1 31718.18,E2 31718.18} C_VEL
LIN {X 0,Y 680.505,Z 200.459,A -85,B 0,C 180,E1 31715.073,E2 31715.073} C_VEL
LIN {X 0,Y 680.52,Z 200.461,A -85,B 0,C 180,E1 31712.133,E2 31712.133} C_VEL
LIN {X 0,Y 680.511,Z 200.453,A -85,B 0,C 180,E1 31709.101,E2 31709.101} C_VEL
LIN {X 0,Y 680.516,Z 200.463,A -85,B 0,C 180,E1 31706.061,E2 31706.061} C_VEL
LIN {X 0,Y 680.511,Z 200.447,A -85,B 0,C 180,E1 31703.007,E2 31703.007} C_VEL
LIN {X 0,Y 680.513,Z 200.459,A -85,B 0,C 180,E1 31700.02,E2 31700.02} C_VEL
LIN {X 0,Y 680.513,Z 200.45,A -85,B 0,C 180,E1 31696.957,E2 31696.957} C_VEL
LIN {X 0,Y 680.508,Z 200.457,A -85,B 0,C 180,E1 31693.944,E2 31693.944} C_VEL
LIN {X 0,Y 680.517,Z 200.45,A -85,B 0,C 180,E1 31690.926,E2 31690.926} C_VEL
LIN {X 0,Y 680.507,Z 200.459,A -85,B 0,C 180,E1 31687.939,E2 31687.939} C_VEL
LIN {X 0,Y 680.518,Z 200.448,A -85,B 0,C 180,E1 31684.889,E2 31684.889} C_VEL
LIN {X 0,Y 680.503,Z 200.46,A -85,B 0,C 180,E1 31681.852,E2 31681.852} C_VEL
LIN {X 0,Y 680.523,Z 200.443,A -85,B 0,C 180,E1 31678.906,E2 31678.906} C_VEL
LIN {X 0,Y 680.503,Z 200.463,A -85,B 0,C 180,E1 31675.871,E2 31675.871} C_VEL
LIN {X 0,Y 680.524,Z 200.444,A -85,B 0,C 180,E1 31672.826,E2 31672.826} C_VEL
LIN {X 0,Y 680.496,Z 200.463,A -85,B 0,C 180,E1 31669.759,E2 31669.759} C_VEL
LIN {X 0,Y 680.525,Z 200.456,A -85,B 0,C 180,E1 31666.749,E2 31666.749} C_VEL
LIN {X 0,Y 680.489,Z 200.464,A -85,B 0,C 180,E1 31663.701,E2 31663.701} C_VEL
LIN {X 0,Y 680.522,Z 200.455,A -85,B 0,C 180,E1 31660.784,E2 31660.784} C_VEL
LIN {X 0,Y 680.49,Z 200.465,A -85,B 0,C 180,E1 31657.722,E2 31657.722} C_VEL
LIN {X 0,Y 680.518,Z 200.457,A -85,B 0,C 180,E1 31654.78,E2 31654.78} C_VEL
LIN {X 0,Y 680.485,Z 200.464,A -85,B 0,C 180,E1 31651.661,E2 31651.661} C_VEL
LIN {X 0,Y 680.516,Z 200.458,A -85,B 0,C 180,E1 31648.757,E2 31648.757} C_VEL
LIN {X 0,Y 680.483,Z 200.466,A -85,B 0,C 180,E1 31645.65,E2 31645.65} C_VEL
LIN {X 0,Y 680.507,Z 200.46,A -85,B 0,C 180,E1 31642.745,E2 31642.745} C_VEL
LIN {X 0,Y 680.486,Z 200.468,A -85,B 0,C 180,E1 31639.694,E2 31639.694} C_VEL
LIN {X 0,Y 680.484,Z 200.463,A -85,B 0,C 180,E1 31636.901,E2 31636.901} C_VEL
LIN {X 0,Y 680.497,Z 200.468,A -85,B 0,C 180,E1 31633.794,E2 31633.794} C_VEL
LIN {X 0,Y 680.546,Z 200.608,A -85,B 0,C 180,E1 31632.351,E2 31632.351} C_VEL
LIN {X 0,Y 681.71,Z 203.762,A -85,B 0,C 180,E1 31632.083,E2 31632.083} C_VEL
LIN {X 0,Y 689.851,Z 220.391,A -85,B 0,C 180,E1 31630.579,E2 31630.579} C_VEL
LIN {X 0,Y 693.4,Z 228.06,A -85,B 0,C 180,E1 31629.945,E2 31629.945} C_VEL
LIN {X 0,Y 691.864,Z 284.655,A -85,B 0,C 180,E1 31627.22,E2 31627.22} C_VEL
LIN {X 0,Y 691.551,Z 300.07,A -85,B 0,C 180,E1 31626.511,E2 31626.511} C_VEL
LIN {X 0,Y 693.628,Z 313.843,A -85,B 0,C 180,E1 31626.236,E2 31626.236} C_VEL
LIN {X 0,Y 691.532,Z 571.069,A -85,B 0,C 180,E1 31623.19,E2 31623.19} C_VEL
LIN {X 0,Y 690.512,Z 691.443,A -85,B 0,C 180,E1 31621.764,E2 31621.764} C_VEL
LIN {X 0,Y 689.975,Z 716.757,A -85,B 0,C 180,E1 31621.316,E2 31621.316} C_VEL
LIN {X 0,Y 689.34,Z 738.451,A -85,B 0,C 180,E1 31620.796,E2 31620.796} C_VEL
LIN {X 0,Y 688.601,Z 762.554,A -85,B 0,C 180,E1 31620.064,E2 31620.064} C_VEL
LIN {X 0,Y 687.791,Z 783.606,A -85,B 0,C 180,E1 31619.277,E2 31619.277} C_VEL
LIN {X 0,Y 686.892,Z 805.964,A -85,B 0,C 180,E1 31618.296,E2 31618.296} C_VEL
LIN {X 0,Y 685.951,Z 827.052,A -85,B 0,C 180,E1 31617.197,E2 31617.197} C_VEL
LIN {X 0,Y 685.062,Z 846.93,A -85,B 0,C 180,E1 31616.013,E2 31616.013} C_VEL
LIN {X 0,Y 684.091,Z 867.293,A -85,B 0,C 180,E1 31614.613,E2 31614.613} C_VEL
LIN {X 0,Y 683.28,Z 885.609,A -85,B 0,C 180,E1 31613.182,E2 31613.182} C_VEL
LIN {X 0,Y 682.485,Z 903.534,A -85,B 0,C 180,E1 31611.576,E2 31611.576} C_VEL
LIN {X 0,Y 681.84,Z 919.628,A -85,B 0,C 180,E1 31609.948,E2 31609.948} C_VEL
LIN {X 0,Y 681.28,Z 934.522,A -85,B 0,C 180,E1 31608.217,E2 31608.217} C_VEL
LIN {X 0,Y 680.844,Z 947.817,A -85,B 0,C 180,E1 31606.463,E2 31606.463} C_VEL
LIN {X 0,Y 680.499,Z 960.282,A -85,B 0,C 180,E1 31604.552,E2 31604.552} C_VEL
LIN {X 0,Y 680.267,Z 970.026,A -85,B 0,C 180,E1 31602.823,E2 31602.823} C_VEL
LIN {X 0,Y 680.079,Z 979.831,A -85,B 0,C 180,E1 31600.762,E2 31600.762} C_VEL
LIN {X 0,Y 679.975,Z 986.817,A -85,B 0,C 180,E1 31598.967,E2 31598.967} C_VEL
LIN {X 0,Y 679.949,Z 993.141,A -85,B 0,C 180,E1 31596.966,E2 31596.966} C_VEL
LIN {X 0,Y 679.895,Z 997.657,A -85,B 0,C 180,E1 31594.978,E2 31594.978} C_VEL
LIN {X 0,Y 679.893,Z 1000.462,A -85,B 0,C 180,E1 31593.204,E2 31593.204} C_VEL
LIN {X 0,Y 679.908,Z 1002.216,A -85,B 0,C 180,E1 31591.095,E2 31591.095} C_VEL
LIN {X 0,Y 679.883,Z 1002.328,A -85,B 0,C 180,E1 31589.326,E2 31589.326} C_VEL
LIN {X 0,Y 679.895,Z 1001.227,A -85,B 0,C 180,E1 31587.471,E2 31587.471} C_VEL
LIN {X 0,Y 679.916,Z 998.29,A -85,B 0,C 180,E1 31585.361,E2 31585.361} C_VEL
LIN {X 0,Y 679.923,Z 994.483,A -85,B 0,C 180,E1 31583.583,E2 31583.583} C_VEL
LIN {X 0,Y 679.965,Z 988.635,A -85,B 0,C 180,E1 31581.544,E2 31581.544} C_VEL
LIN {X 0,Y 680.074,Z 981.384,A -85,B 0,C 180,E1 31579.613,E2 31579.613} C_VEL
LIN {X 0,Y 680.222,Z 972.709,A -85,B 0,C 180,E1 31577.693,E2 31577.693} C_VEL
LIN {X 0,Y 680.456,Z 961.84,A -85,B 0,C 180,E1 31575.708,E2 31575.708} C_VEL
LIN {X 0,Y 680.777,Z 950.047,A -85,B 0,C 180,E1 31573.856,E2 31573.856} C_VEL
LIN {X 0,Y 681.229,Z 935.929,A -85,B 0,C 180,E1 31571.959,E2 31571.959} C_VEL
LIN {X 0,Y 681.78,Z 920.971,A -85,B 0,C 180,E1 31570.197,E2 31570.197} C_VEL
LIN {X 0,Y 682.449,Z 904.46,A -85,B 0,C 180,E1 31568.513,E2 31568.513} C_VEL
LIN {X 0,Y 683.235,Z 886.712,A -85,B 0,C 180,E1 31566.908,E2 31566.908} C_VEL
LIN {X 0,Y 684.071,Z 867.771,A -85,B 0,C 180,E1 31565.423,E2 31565.423} C_VEL
LIN {X 0,Y 685.031,Z 847.628,A -85,B 0,C 180,E1 31564.031,E2 31564.031} C_VEL
LIN {X 0,Y 685.913,Z 827.937,A -85,B 0,C 180,E1 31562.853,E2 31562.853} C_VEL
LIN {X 0,Y 686.869,Z 806.495,A -85,B 0,C 180,E1 31561.729,E2 31561.729} C_VEL
LIN {X 0,Y 687.759,Z 784.48,A -85,B 0,C 180,E1 31560.759,E2 31560.759} C_VEL
LIN {X 0,Y 688.548,Z 763.835,A -85,B 0,C 180,E1 31559.982,E2 31559.982} C_VEL
LIN {X 0,Y 689.331,Z 738.773,A -85,B 0,C 180,E1 31559.213,E2 31559.213} C_VEL
LIN {X 0,Y 689.962,Z 717.146,A -85,B 0,C 180,E1 31558.693,E2 31558.693} C_VEL
LIN {X 0,Y 690.509,Z 691.704,A -85,B 0,C 180,E1 31558.24,E2 31558.24} C_VEL
LIN {X 0,Y 691.408,Z 586.497,A -85,B 0,C 180,E1 31556.991,E2 31556.991} C_VEL
LIN {X 0,Y 693.602,Z 318.417,A -85,B 0,C 180,E1 31553.817,E2 31553.817} C_VEL
LIN {X 0,Y 693.37,Z 310.96,A -85,B 0,C 180,E1 31553.719,E2 31553.719} C_VEL
LIN {X 0,Y 691.268,Z 298.667,A -85,B 0,C 180,E1 31553.472,E2 31553.472} C_VEL
LIN {X 0,Y 691.963,Z 260.145,A -85,B 0,C 180,E1 31551.688,E2 31551.688} C_VEL
LIN {X 0,Y 693.257,Z 227.855,A -85,B 0,C 180,E1 31550.072,E2 31550.072} C_VEL
LIN {X 0,Y 686.717,Z 213.41,A -85,B 0,C 180,E1 31548.674,E2 31548.674} C_VEL
LIN {X 0,Y 682.333,Z 204.616,A -85,B 0,C 180,E1 31547.609,E2 31547.609} C_VEL
LIN {X 0,Y 680.649,Z 201.213,A -85,B 0,C 180,E1 31547.143,E2 31547.143} C_VEL
LIN {X 0,Y 680.521,Z 200.466,A -85,B 0,C 180,E1 31547.019,E2 31547.019} C_VEL
LIN {X 0,Y 680.507,Z 200.467,A -85,B 0,C 180,E1 31544.027,E2 31544.027} C_VEL
LIN {X 0,Y 680.523,Z 200.466,A -85,B 0,C 180,E1 31540.955,E2 31540.955} C_VEL
LIN {X 0,Y 680.524,Z 200.466,A -85,B 0,C 180,E1 31537.891,E2 31537.891} C_VEL
LIN {X 0,Y 680.554,Z 200.698,A -85,B 0,C 180,E1 31536.74,E2 31536.74} C_VEL
LIN {X 0,Y 682.051,Z 204.299,A -85,B 0,C 180,E1 31536.264,E2 31536.264} C_VEL
LIN {X 0,Y 685.777,Z 212.313,A -85,B 0,C 180,E1 31535.264,E2 31535.264} C_VEL
LIN {X 0,Y 690.176,Z 223.8,A -85,B 0,C 180,E1 31534.066,E2 31534.066} C_VEL
LIN {X 0,Y 687.73,Z 268.398,A -85,B 0,C 180,E1 31531.252,E2 31531.252} C_VEL
LIN {X 0,Y 685.83,Z 323.875,A -85,B 0,C 180,E1 31527.932,E2 31527.932} C_VEL
LIN {X 0,Y 684.59,Z 376.896,A -85,B 0,C 180,E1 31524.875,E2 31524.875} C_VEL
LIN {X 0,Y 683.539,Z 431.477,A -85,B 0,C 180,E1 31521.812,E2 31521.812} C_VEL
LIN {X 0,Y 683.134,Z 459.994,A -85,B 0,C 180,E1 31520.256,E2 31520.256} C_VEL
LIN {X 0,Y 685.436,Z 480.384,A -85,B 0,C 180,E1 31519.869,E2 31519.869} C_VEL
LIN {X 0,Y 683.692,Z 621.003,A -85,B 0,C 180,E1 31518.146,E2 31518.146} C_VEL
LIN {X 0,Y 683.238,Z 681.836,A -85,B 0,C 180,E1 31517.414,E2 31517.414} C_VEL
LIN {X 0,Y 682.981,Z 701.179,A -85,B 0,C 180,E1 31517.026,E2 31517.026} C_VEL
LIN {X 0,Y 682.68,Z 719.393,A -85,B 0,C 180,E1 31516.508,E2 31516.508} C_VEL
LIN {X 0,Y 682.322,Z 736.765,A -85,B 0,C 180,E1 31515.861,E2 31515.861} C_VEL
LIN {X 0,Y 681.971,Z 752.982,A -85,B 0,C 180,E1 31515.103,E2 31515.103} C_VEL
LIN {X 0,Y 681.609,Z 768.373,A -85,B 0,C 180,E1 31514.224,E2 31514.224} C_VEL
LIN {X 0,Y 681.227,Z 783.257,A -85,B 0,C 180,E1 31513.194,E2 31513.194} C_VEL
LIN {X 0,Y 680.897,Z 796.161,A -85,B 0,C 180,E1 31512.122,E2 31512.122} C_VEL
LIN {X 0,Y 680.603,Z 808.196,A -85,B 0,C 180,E1 31510.925,E2 31510.925} C_VEL
LIN {X 0,Y 680.352,Z 818.873,A -85,B 0,C 180,E1 31509.645,E2 31509.645} C_VEL
LIN {X 0,Y 680.158,Z 828.192,A -85,B 0,C 180,E1 31508.283,E2 31508.283} C_VEL
LIN {X 0,Y 680.025,Z 836.118,A -85,B 0,C 180,E1 31506.84,E2 31506.84} C_VEL
LIN {X 0,Y 679.955,Z 842.584,A -85,B 0,C 180,E1 31505.316,E2 31505.316} C_VEL
LIN {X 0,Y 679.922,Z 847.646,A -85,B 0,C 180,E1 31503.71,E2 31503.71} C_VEL
LIN {X 0,Y 679.911,Z 850.776,A -85,B 0,C 180,E1 31502.191,E2 31502.191} C_VEL
LIN {X 0,Y 679.915,Z 852.336,A -85,B 0,C 180,E1 31500.59,E2 31500.59} C_VEL
LIN {X 0,Y 679.918,Z 852.154,A -85,B 0,C 180,E1 31498.989,E2 31498.989} C_VEL
LIN {X 0,Y 679.916,Z 850.224,A -85,B 0,C 180,E1 31497.387,E2 31497.387} C_VEL
LIN {X 0,Y 679.922,Z 846.748,A -85,B 0,C 180,E1 31495.868,E2 31495.868} C_VEL
LIN {X 0,Y 679.958,Z 841.259,A -85,B 0,C 180,E1 31494.261,E2 31494.261} C_VEL
LIN {X 0,Y 680.045,Z 834.309,A -85,B 0,C 180,E1 31492.736,E2 31492.736} C_VEL
LIN {X 0,Y 680.178,Z 825.862,A -85,B 0,C 180,E1 31491.291,E2 31491.291} C_VEL
LIN {X 0,Y 680.396,Z 815.288,A -85,B 0,C 180,E1 31489.843,E2 31489.843} C_VEL
LIN {X 0,Y 680.654,Z 803.831,A -85,B 0,C 180,E1 31488.561,E2 31488.561} C_VEL
LIN {X 0,Y 680.984,Z 790.402,A -85,B 0,C 180,E1 31487.32,E2 31487.32} C_VEL
LIN {X 0,Y 681.352,Z 775.779,A -85,B 0,C 180,E1 31486.204,E2 31486.204} C_VEL
LIN {X 0,Y 681.746,Z 760.057,A -85,B 0,C 180,E1 31485.215,E2 31485.215} C_VEL
LIN {X 0,Y 682.118,Z 743.276,A -85,B 0,C 180,E1 31484.352,E2 31484.352} C_VEL
LIN {X 0,Y 682.53,Z 725.39,A -85,B 0,C 180,E1 31483.62,E2 31483.62} C_VEL
LIN {X 0,Y 682.868,Z 706.517,A -85,B 0,C 180,E1 31483.029,E2 31483.029} C_VEL
LIN {X 0,Y 683.139,Z 687.496,A -85,B 0,C 180,E1 31482.602,E2 31482.602} C_VEL
LIN {X 0,Y 683.329,Z 666.69,A -85,B 0,C 180,E1 31482.308,E2 31482.308} C_VEL
LIN {X 0,Y 683.666,Z 595.646,A -85,B 0,C 180,E1 31481.524,E2 31481.524} C_VEL
LIN {X 0,Y 682.791,Z 588.053,A -85,B 0,C 180,E1 31481.408,E2 31481.408} C_VEL
LIN {X 0,Y 677.088,Z 568.181,A -85,B 0,C 180,E1 31480.994,E2 31480.994} C_VEL
LIN {X 0,Y 676.454,Z 561.656,A -85,B 0,C 180,E1 31480.895,E2 31480.895} C_VEL
LIN {X 0,Y 676.947,Z 477.791,A -85,B 0,C 180,E1 31479.914,E2 31479.914} C_VEL
LIN {X 0,Y 675.482,Z 465.394,A -85,B 0,C 180,E1 31479.689,E2 31479.689} C_VEL
LIN {X 0,Y 676.601,Z 409.918,A -85,B 0,C 180,E1 31476.576,E2 31476.576} C_VEL
LIN {X 0,Y 677.746,Z 356.691,A -85,B 0,C 180,E1 31473.542,E2 31473.542} C_VEL
LIN {X 0,Y 679.018,Z 304.926,A -85,B 0,C 180,E1 31470.539,E2 31470.539} C_VEL
LIN {X 0,Y 680.442,Z 252.93,A -85,B 0,C 180,E1 31467.464,E2 31467.464} C_VEL
LIN {X 0,Y 681.13,Z 224.316,A -85,B 0,C 180,E1 31465.739,E2 31465.739} C_VEL
LIN {X 0,Y 672.579,Z 201.441,A -85,B 0,C 180,E1 31463.805,E2 31463.805} C_VEL
LIN {X 0,Y 672.545,Z 201.456,A -85,B 0,C 180,E1 31460.902,E2 31460.902} C_VEL
LIN {X 0,Y 672.529,Z 201.456,A -85,B 0,C 180,E1 31457.892,E2 31457.892} C_VEL
LIN {X 0,Y 672.582,Z 201.45,A -85,B 0,C 180,E1 31455.044,E2 31455.044} C_VEL
LIN {X 0,Y 672.588,Z 201.453,A -85,B 0,C 180,E1 31451.985,E2 31451.985} C_VEL
LIN {X 0,Y 672.513,Z 201.456,A -85,B 0,C 180,E1 31449.19,E2 31449.19} C_VEL
LIN {X 0,Y 672.579,Z 201.622,A -85,B 0,C 180,E1 31446.887,E2 31446.887} C_VEL
LIN {X 0,Y 679.346,Z 218.804,A -85,B 0,C 180,E1 31445.307,E2 31445.307} C_VEL
LIN {X 0,Y 682.037,Z 226.59,A -85,B 0,C 180,E1 31444.566,E2 31444.566} C_VEL
LIN {X 0,Y 680.752,Z 266.781,A -85,B 0,C 180,E1 31441.625,E2 31441.625} C_VEL
LIN {X 0,Y 679.52,Z 306.415,A -85,B 0,C 180,E1 31438.762,E2 31438.762} C_VEL
LIN {X 0,Y 679.485,Z 310.379,A -85,B 0,C 180,E1 31438.496,E2 31438.496} C_VEL
LIN {X 0,Y 681.228,Z 320.364,A -85,B 0,C 180,E1 31438.294,E2 31438.294} C_VEL
LIN {X 0,Y 679.45,Z 568.033,A -85,B 0,C 180,E1 31435.484,E2 31435.484} C_VEL
LIN {X 0,Y 679.106,Z 608.658,A -85,B 0,C 180,E1 31435,E2 31435} C_VEL
LIN {X 0,Y 678.694,Z 631.405,A -85,B 0,C 180,E1 31434.586,E2 31434.586} C_VEL
LIN {X 0,Y 678.15,Z 652.378,A -85,B 0,C 180,E1 31434.036,E2 31434.036} C_VEL
LIN {X 0,Y 677.64,Z 669.474,A -85,B 0,C 180,E1 31433.478,E2 31433.478} C_VEL
LIN {X 0,Y 677.053,Z 686.549,A -85,B 0,C 180,E1 31432.81,E2 31432.81} C_VEL
LIN {X 0,Y 676.5,Z 702.61,A -85,B 0,C 180,E1 31432.069,E2 31432.069} C_VEL
LIN {X 0,Y 675.912,Z 718.028,A -85,B 0,C 180,E1 31431.25,E2 31431.25} C_VEL
LIN {X 0,Y 675.272,Z 734.049,A -85,B 0,C 180,E1 31430.273,E2 31430.273} C_VEL
LIN {X 0,Y 674.601,Z 751.677,A -85,B 0,C 180,E1 31429.031,E2 31429.031} C_VEL
LIN {X 0,Y 673.925,Z 768.647,A -85,B 0,C 180,E1 31427.618,E2 31427.618} C_VEL
LIN {X 0,Y 673.437,Z 781.527,A -85,B 0,C 180,E1 31426.386,E2 31426.386} C_VEL
LIN {X 0,Y 673.036,Z 793.645,A -85,B 0,C 180,E1 31425.069,E2 31425.069} C_VEL
LIN {X 0,Y 672.65,Z 806.255,A -85,B 0,C 180,E1 31423.496,E2 31423.496} C_VEL
LIN {X 0,Y 672.335,Z 818.497,A -85,B 0,C 180,E1 31421.669,E2 31421.669} C_VEL
LIN {X 0,Y 672.156,Z 827.245,A -85,B 0,C 180,E1 31420.11,E2 31420.11} C_VEL
